LIN {X 0,Y 362.034,Z 645.085,A -85,B 0,C 180,E1 -21360.313,E2 -21360.313} C_VEL
LIN {X 0,Y 359.449,Z 640.545,A -85,B 0,C 180,E1 -21361.106,E2 -21361.106} C_VEL
LIN {X 0,Y 359.251,Z 639.964,A -85,B 0,C 180,E1 -21361.22,E2 -21361.22} C_VEL
LIN {X 0,Y 357.675,Z 633.23,A -85,B 0,C 180,E1 -21364.664,E2 -21364.664} C_VEL
LIN {X 0,Y 356.244,Z 627.609,A -85,B 0,C 180,E1 -21368.142,E2 -21368.142} C_VEL
LIN {X 0,Y 354.982,Z 623.589,A -85,B 0,C 180,E1 -21371.426,E2 -21371.426} C_VEL
LIN {X 0,Y 354.115,Z 620.735,A -85,B 0,C 180,E1 -21374.595,E2 -21374.595} C_VEL
LIN {X 0,Y 353.624,Z 618.917,A -85,B 0,C 180,E1 -21377.665,E2 -21377.665} C_VEL
LIN {X 0,Y 353.31,Z 618.175,A -85,B 0,C 180,E1 -21380.641,E2 -21380.641} C_VEL
LIN {X 0,Y 353.46,Z 618.481,A -85,B 0,C 180,E1 -21384.34,E2 -21384.34} C_VEL
LIN {X 0,Y 353.86,Z 619.974,A -85,B 0,C 180,E1 -21387.693,E2 -21387.693} C_VEL
LIN {X 0,Y 354.531,Z 621.978,A -85,B 0,C 180,E1 -21390.401,E2 -21390.401} C_VEL
LIN {X 0,Y 355.324,Z 624.648,A -85,B 0,C 180,E1 -21393.038,E2 -21393.038} C_VEL
LIN {X 0,Y 356.135,Z 627.934,A -85,B 0,C 180,E1 -21395.605,E2 -21395.605} C_VEL
LIN {X 0,Y 357.351,Z 632.416,A -85,B 0,C 180,E1 -21398.474,E2 -21398.474} C_VEL
LIN {X 0,Y 359.745,Z 636.348,A -85,B 0,C 180,E1 -21399.232,E2 -21399.232} C_VEL
LIN {X 0,Y 361.184,Z 638.274,A -85,B 0,C 180,E1 -21399.647,E2 -21399.647} C_VEL
LIN {X 0,Y 364.586,Z 643.755,A -85,B 0,C 180,E1 -21400.618,E2 -21400.618} C_VEL
LIN {X 0,Y 369.272,Z 651.818,A -85,B 0,C 180,E1 -21401.891,E2 -21401.891} C_VEL
LIN {X 0,Y 374.557,Z 662.104,A -85,B 0,C 180,E1 -21403.232,E2 -21403.232} C_VEL
LIN {X 0,Y 377.698,Z 669.576,A -85,B 0,C 180,E1 -21404.051,E2 -21404.051} C_VEL
LIN {X 0,Y 378.425,Z 674.581,A -85,B 0,C 180,E1 -21404.369,E2 -21404.369} C_VEL
LIN {X 0,Y 373.198,Z 737.25,A -85,B 0,C 180,E1 -21406.258,E2 -21406.258} C_VEL
LIN {X 0,Y 372.142,Z 747.157,A -85,B 0,C 180,E1 -21406.669,E2 -21406.669} C_VEL
LIN {X 0,Y 370.881,Z 756.699,A -85,B 0,C 180,E1 -21407.178,E2 -21407.178} C_VEL
LIN {X 0,Y 369.456,Z 766.257,A -85,B 0,C 180,E1 -21407.824,E2 -21407.824} C_VEL
LIN {X 0,Y 367.532,Z 777.167,A -85,B 0,C 180,E1 -21408.735,E2 -21408.735} C_VEL
LIN {X 0,Y 365.707,Z 786.264,A -85,B 0,C 180,E1 -21409.656,E2 -21409.656} C_VEL
LIN {X 0,Y 364.062,Z 793.981,A -85,B 0,C 180,E1 -21410.587,E2 -21410.587} C_VEL
LIN {X 0,Y 362.212,Z 801.591,A -85,B 0,C 180,E1 -21411.66,E2 -21411.66} C_VEL
LIN {X 0,Y 360.099,Z 809.415,A -85,B 0,C 180,E1 -21412.984,E2 -21412.984} C_VEL
LIN {X 0,Y 358.035,Z 816.293,A -85,B 0,C 180,E1 -21414.386,E2 -21414.386} C_VEL
LIN {X 0,Y 356.572,Z 820.935,A -85,B 0,C 180,E1 -21415.493,E2 -21415.493} C_VEL
LIN {X 0,Y 354.669,Z 826.661,A -85,B 0,C 180,E1 -21417.17,E2 -21417.17} C_VEL
LIN {X 0,Y 353.04,Z 831.154,A -85,B 0,C 180,E1 -21418.863,E2 -21418.863} C_VEL
LIN {X 0,Y 352.202,Z 833.462,A -85,B 0,C 180,E1 -21420,E2 -21420} C_VEL
LIN {X 0,Y 350.875,Z 836.886,A -85,B 0,C 180,E1 -21422.288,E2 -21422.288} C_VEL
LIN {X 0,Y 349.954,Z 838.441,A -85,B 0,C 180,E1 -21424.592,E2 -21424.592} C_VEL
LIN {X 0,Y 349.611,Z 838.707,A -85,B 0,C 180,E1 -21425.749,E2 -21425.749} C_VEL
LIN {X 0,Y 349.177,Z 837.732,A -85,B 0,C 180,E1 -21428.072,E2 -21428.072} C_VEL
LIN {X 0,Y 349.123,Z 836.645,A -85,B 0,C 180,E1 -21429.236,E2 -21429.236} C_VEL
LIN {X 0,Y 349.169,Z 834.725,A -85,B 0,C 180,E1 -21430.592,E2 -21430.592} C_VEL
LIN {X 0,Y 349.117,Z 831.765,A -85,B 0,C 180,E1 -21432.161,E2 -21432.161} C_VEL
LIN {X 0,Y 349.316,Z 827.362,A -85,B 0,C 180,E1 -21433.923,E2 -21433.923} C_VEL
LIN {X 0,Y 349.612,Z 822.276,A -85,B 0,C 180,E1 -21435.516,E2 -21435.516} C_VEL
LIN {X 0,Y 349.838,Z 816.988,A -85,B 0,C 180,E1 -21436.877,E2 -21436.877} C_VEL
LIN {X 0,Y 350.091,Z 811.586,A -85,B 0,C 180,E1 -21438.066,E2 -21438.066} C_VEL
LIN {X 0,Y 350.483,Z 805.301,A -85,B 0,C 180,E1 -21439.253,E2 -21439.253} C_VEL
LIN {X 0,Y 350.964,Z 797.406,A -85,B 0,C 180,E1 -21440.512,E2 -21440.512} C_VEL
LIN {X 0,Y 351.517,Z 787.781,A -85,B 0,C 180,E1 -21441.785,E2 -21441.785} C_VEL
LIN {X 0,Y 352.089,Z 778.326,A -85,B 0,C 180,E1 -21442.825,E2 -21442.825} C_VEL
LIN {X 0,Y 352.732,Z 767.619,A -85,B 0,C 180,E1 -21443.791,E2 -21443.791} C_VEL
LIN {X 0,Y 353.212,Z 757.652,A -85,B 0,C 180,E1 -21444.521,E2 -21444.521} C_VEL
LIN {X 0,Y 353.539,Z 747.147,A -85,B 0,C 180,E1 -21445.133,E2 -21445.133} C_VEL
LIN {X 0,Y 353.943,Z 736.192,A -85,B 0,C 180,E1 -21445.612,E2 -21445.612} C_VEL
LIN {X 0,Y 354.734,Z 713.298,A -85,B 0,C 180,E1 -21446.298,E2 -21446.298} C_VEL
LIN {X 0,Y 356.077,Z 658.366,A -85,B 0,C 180,E1 -21447.873,E2 -21447.873} C_VEL
LIN {X 0,Y 353.084,Z 631.016,A -85,B 0,C 180,E1 -21448.746,E2 -21448.746} C_VEL
LIN {X 0,Y 352.843,Z 627.653,A -85,B 0,C 180,E1 -21448.863,E2 -21448.863} C_VEL
LIN {X 0,Y 353.374,Z 621.195,A -85,B 0,C 180,E1 -21450.69,E2 -21450.69} C_VEL
LIN {X 0,Y 352.052,Z 613.561,A -85,B 0,C 180,E1 -21452.992,E2 -21452.992} C_VEL
LIN {X 0,Y 351.912,Z 613.577,A -85,B 0,C 180,E1 -21457.235,E2 -21457.235} C_VEL
LIN {X 0,Y 351.881,Z 613.582,A -85,B 0,C 180,E1 -21461.062,E2 -21461.062} C_VEL
LIN {X 0,Y 351.929,Z 613.579,A -85,B 0,C 180,E1 -21464.233,E2 -21464.233} C_VEL
LIN {X 0,Y 351.919,Z 613.577,A -85,B 0,C 180,E1 -21467.427,E2 -21467.427} C_VEL
LIN {X 0,Y 351.872,Z 613.583,A -85,B 0,C 180,E1 -21470.926,E2 -21470.926} C_VEL
LIN {X 0,Y 351.907,Z 613.579,A -85,B 0,C 180,E1 -21473.335,E2 -21473.335} C_VEL
LIN {X 0,Y 351.883,Z 613.581,A -85,B 0,C 180,E1 -21476.723,E2 -21476.723} C_VEL
LIN {X 0,Y 351.923,Z 613.582,A -85,B 0,C 180,E1 -21480.159,E2 -21480.159} C_VEL
LIN {X 0,Y 351.926,Z 613.578,A -85,B 0,C 180,E1 -21483.59,E2 -21483.59} C_VEL
LIN {X 0,Y 351.975,Z 613.571,A -85,B 0,C 180,E1 -21486.546,E2 -21486.546} C_VEL
LIN {X 0,Y 351.959,Z 613.576,A -85,B 0,C 180,E1 -21490.225,E2 -21490.225} C_VEL
LIN {X 0,Y 352.021,Z 613.569,A -85,B 0,C 180,E1 -21493.825,E2 -21493.825} C_VEL
LIN {X 0,Y 352.11,Z 613.554,A -85,B 0,C 180,E1 -21497.36,E2 -21497.36} C_VEL
LIN {X 0,Y 352.152,Z 613.549,A -85,B 0,C 180,E1 -21500.844,E2 -21500.844} C_VEL
LIN {X 0,Y 352.258,Z 613.537,A -85,B 0,C 180,E1 -21504.294,E2 -21504.294} C_VEL
LIN {X 0,Y 352.315,Z 613.531,A -85,B 0,C 180,E1 -21507.721,E2 -21507.721} C_VEL
LIN {X 0,Y 352.255,Z 613.536,A -85,B 0,C 180,E1 -21511.139,E2 -21511.139} C_VEL
LIN {X 0,Y 352.328,Z 613.526,A -85,B 0,C 180,E1 -21514.561,E2 -21514.561} C_VEL
LIN {X 0,Y 352.244,Z 613.537,A -85,B 0,C 180,E1 -21516.852,E2 -21516.852} C_VEL
LIN {X 0,Y 352.1,Z 613.558,A -85,B 0,C 180,E1 -21520.314,E2 -21520.314} C_VEL
LIN {X 0,Y 352.044,Z 613.565,A -85,B 0,C 180,E1 -21523.813,E2 -21523.813} C_VEL
LIN {X 0,Y 352.014,Z 613.566,A -85,B 0,C 180,E1 -21527.366,E2 -21527.366} C_VEL
LIN {X 0,Y 351.956,Z 613.573,A -85,B 0,C 180,E1 -21530.991,E2 -21530.991} C_VEL
LIN {X 0,Y 351.941,Z 613.577,A -85,B 0,C 180,E1 -21533.724,E2 -21533.724} C_VEL
LIN {X 0,Y 351.908,Z 613.579,A -85,B 0,C 180,E1 -21537.245,E2 -21537.245} C_VEL
LIN {X 0,Y 351.926,Z 613.581,A -85,B 0,C 180,E1 -21539.84,E2 -21539.84} C_VEL
LIN {X 0,Y 351.92,Z 613.581,A -85,B 0,C 180,E1 -21543.869,E2 -21543.869} C_VEL
LIN {X 0,Y 351.953,Z 613.573,A -85,B 0,C 180,E1 -21547.245,E2 -21547.245} C_VEL
LIN {X 0,Y 351.92,Z 613.577,A -85,B 0,C 180,E1 -21551.057,E2 -21551.057} C_VEL
LIN {X 0,Y 351.927,Z 613.579,A -85,B 0,C 180,E1 -21554.234,E2 -21554.234} C_VEL
LIN {X 0,Y 351.918,Z 613.578,A -85,B 0,C 180,E1 -21557.428,E2 -21557.428} C_VEL
LIN {X 0,Y 351.899,Z 613.58,A -85,B 0,C 180,E1 -21560.921,E2 -21560.921} C_VEL
LIN {X 0,Y 351.933,Z 613.575,A -85,B 0,C 180,E1 -21564.688,E2 -21564.688} C_VEL
LIN {X 0,Y 351.92,Z 613.577,A -85,B 0,C 180,E1 -21568.853,E2 -21568.853} C_VEL
LIN {X 0,Y 351.96,Z 613.573,A -85,B 0,C 180,E1 -21571.47,E2 -21571.47} C_VEL
LIN {X 0,Y 351.9,Z 613.58,A -85,B 0,C 180,E1 -21575.292,E2 -21575.292} C_VEL
LIN {X 0,Y 351.907,Z 613.583,A -85,B 0,C 180,E1 -21577.78,E2 -21577.78} C_VEL
LIN {X 0,Y 351.958,Z 613.576,A -85,B 0,C 180,E1 -21580.226,E2 -21580.226} C_VEL
LIN {X 0,Y 351.98,Z 613.573,A -85,B 0,C 180,E1 -21583.824,E2 -21583.824} C_VEL
LIN {X 0,Y 352.108,Z 613.555,A -85,B 0,C 180,E1 -21587.361,E2 -21587.361} C_VEL
LIN {X 0,Y 352.156,Z 613.547,A -85,B 0,C 180,E1 -21590.845,E2 -21590.845} C_VEL
LIN {X 0,Y 352.3,Z 613.533,A -85,B 0,C 180,E1 -21594.295,E2 -21594.295} C_VEL
LIN {X 0,Y 352.319,Z 613.531,A -85,B 0,C 180,E1 -21597.722,E2 -21597.722} C_VEL
LIN {X 0,Y 352.255,Z 613.535,A -85,B 0,C 180,E1 -21601.14,E2 -21601.14} C_VEL
LIN {X 0,Y 352.327,Z 613.528,A -85,B 0,C 180,E1 -21604.561,E2 -21604.561} C_VEL
LIN {X 0,Y 352.248,Z 613.537,A -85,B 0,C 180,E1 -21606.853,E2 -21606.853} C_VEL
LIN {X 0,Y 352.181,Z 613.551,A -85,B 0,C 180,E1 -21608.003,E2 -21608.003} C_VEL
LIN {X 0,Y 351.48,Z 613.633,A -85,B 0,C 180,E1 -21608.957,E2 -21608.957} C_VEL
LIN {X 0,Y 348.656,Z 613.984,A -85,B 0,C 180,E1 -21610.508,E2 -21610.508} C_VEL
LIN {X 0,Y 346.248,Z 614.287,A -85,B 0,C 180,E1 -21611.763,E2 -21611.763} C_VEL
LIN {X 0,Y 345.156,Z 614.419,A -85,B 0,C 180,E1 -21612.733,E2 -21612.733} C_VEL
LIN {X 0,Y 345.035,Z 614.434,A -85,B 0,C 180,E1 -21613.062,E2 -21613.062} C_VEL
LIN {X 0,Y 344.905,Z 614.452,A -85,B 0,C 180,E1 -21617.352,E2 -21617.352} C_VEL
LIN {X 0,Y 344.874,Z 614.454,A -85,B 0,C 180,E1 -21620.89,E2 -21620.89} C_VEL
LIN {X 0,Y 344.883,Z 614.459,A -85,B 0,C 180,E1 -21623.966,E2 -21623.966} C_VEL
LIN {X 0,Y 344.893,Z 614.457,A -85,B 0,C 180,E1 -21627.847,E2 -21627.847} C_VEL
LIN {X 0,Y 344.816,Z 614.462,A -85,B 0,C 180,E1 -21631.442,E2 -21631.442} C_VEL
LIN {X 0,Y 344.834,Z 614.461,A -85,B 0,C 180,E1 -21634.663,E2 -21634.663} C_VEL
LIN {X 0,Y 344.854,Z 614.46,A -85,B 0,C 180,E1 -21637.614,E2 -21637.614} C_VEL
LIN {X 0,Y 344.822,Z 614.46,A -85,B 0,C 180,E1 -21641.272,E2 -21641.272} C_VEL
LIN {X 0,Y 344.799,Z 614.465,A -85,B 0,C 180,E1 -21644.683,E2 -21644.683} C_VEL
LIN {X 0,Y 344.817,Z 614.467,A -85,B 0,C 180,E1 -21647.907,E2 -21647.907} C_VEL
LIN {X 0,Y 344.81,Z 614.461,A -85,B 0,C 180,E1 -21650.97,E2 -21650.97} C_VEL
LIN {X 0,Y 344.821,Z 614.464,A -85,B 0,C 180,E1 -21654.344,E2 -21654.344} C_VEL
LIN {X 0,Y 344.826,Z 614.461,A -85,B 0,C 180,E1 -21656.739,E2 -21656.739} C_VEL
LIN {X 0,Y 344.833,Z 614.458,A -85,B 0,C 180,E1 -21660.824,E2 -21660.824} C_VEL
LIN {X 0,Y 344.968,Z 614.643,A -85,B 0,C 180,E1 -21663.175,E2 -21663.175} C_VEL
LIN {X 0,Y 347.071,Z 626.547,A -85,B 0,C 180,E1 -21666.51,E2 -21666.51} C_VEL
LIN {X 0,Y 347.053,Z 630.044,A -85,B 0,C 180,E1 -21667.451,E2 -21667.451} C_VEL
LIN {X 0,Y 345.418,Z 643.632,A -85,B 0,C 180,E1 -21670.991,E2 -21670.991} C_VEL
LIN {X 0,Y 347.217,Z 668.999,A -85,B 0,C 180,E1 -21671.803,E2 -21671.803} C_VEL
LIN {X 0,Y 348.767,Z 684.999,A -85,B 0,C 180,E1 -21672.312,E2 -21672.312} C_VEL
LIN {X 0,Y 347.023,Z 749.499,A -85,B 0,C 180,E1 -21674.225,E2 -21674.225} C_VEL
LIN {X 0,Y 346.578,Z 759.945,A -85,B 0,C 180,E1 -21674.655,E2 -21674.655} C_VEL
LIN {X 0,Y 346.235,Z 769.907,A -85,B 0,C 180,E1 -21675.202,E2 -21675.202} C_VEL
LIN {X 0,Y 345.748,Z 780.31,A -85,B 0,C 180,E1 -21675.93,E2 -21675.93} C_VEL
LIN {X 0,Y 345.259,Z 789.479,A -85,B 0,C 180,E1 -21676.716,E2 -21676.716} C_VEL
LIN {X 0,Y 344.524,Z 799.727,A -85,B 0,C 180,E1 -21677.789,E2 -21677.789} C_VEL
LIN {X 0,Y 344.029,Z 808.158,A -85,B 0,C 180,E1 -21678.848,E2 -21678.848} C_VEL
LIN {X 0,Y 343.55,Z 816.054,A -85,B 0,C 180,E1 -21680.02,E2 -21680.02} C_VEL
LIN {X 0,Y 343.024,Z 824.278,A -85,B 0,C 180,E1 -21681.487,E2 -21681.487} C_VEL
LIN {X 0,Y 342.777,Z 831.149,A -85,B 0,C 180,E1 -21682.958,E2 -21682.958} C_VEL
LIN {X 0,Y 342.591,Z 835.863,A -85,B 0,C 180,E1 -21684.133,E2 -21684.133} C_VEL
LIN {X 0,Y 342.46,Z 841.572,A -85,B 0,C 180,E1 -21685.895,E2 -21685.895} C_VEL
LIN {X 0,Y 342.421,Z 846.02,A -85,B 0,C 180,E1 -21687.656,E2 -21687.656} C_VEL
LIN {X 0,Y 342.371,Z 848.381,A -85,B 0,C 180,E1 -21688.828,E2 -21688.828} C_VEL
LIN {X 0,Y 342.277,Z 851.57,A -85,B 0,C 180,E1 -21691.173,E2 -21691.173} C_VEL
LIN {X 0,Y 342.251,Z 852.514,A -85,B 0,C 180,E1 -21692.346,E2 -21692.346} C_VEL
LIN {X 0,Y 342.314,Z 853.154,A -85,B 0,C 180,E1 -21694.695,E2 -21694.695} C_VEL
LIN {X 0,Y 342.824,Z 852.017,A -85,B 0,C 180,E1 -21697.042,E2 -21697.042} C_VEL
LIN {X 0,Y 343.184,Z 850.939,A -85,B 0,C 180,E1 -21698.214,E2 -21698.214} C_VEL
LIN {X 0,Y 344.459,Z 847.292,A -85,B 0,C 180,E1 -21700.545,E2 -21700.545} C_VEL
LIN {X 0,Y 345.803,Z 843.392,A -85,B 0,C 180,E1 -21702.28,E2 -21702.28} C_VEL
LIN {X 0,Y 347.54,Z 838.373,A -85,B 0,C 180,E1 -21703.996,E2 -21703.996} C_VEL
LIN {X 0,Y 349.51,Z 832.307,A -85,B 0,C 180,E1 -21705.651,E2 -21705.651} C_VEL
LIN {X 0,Y 351.436,Z 825.979,A -85,B 0,C 180,E1 -21707.067,E2 -21707.067} C_VEL
LIN {X 0,Y 353.704,Z 818.316,A -85,B 0,C 180,E1 -21708.473,E2 -21708.473} C_VEL
LIN {X 0,Y 356.07,Z 809.306,A -85,B 0,C 180,E1 -21709.837,E2 -21709.837} C_VEL
LIN {X 0,Y 358.245,Z 800.757,A -85,B 0,C 180,E1 -21710.906,E2 -21710.906} C_VEL
LIN {X 0,Y 360.206,Z 792.083,A -85,B 0,C 180,E1 -21711.833,E2 -21711.833} C_VEL
LIN {X 0,Y 362.445,Z 781.582,A -85,B 0,C 180,E1 -21712.738,E2 -21712.738} C_VEL
LIN {X 0,Y 364.311,Z 771.526,A -85,B 0,C 180,E1 -21713.438,E2 -21713.438} C_VEL
LIN {X 0,Y 365.885,Z 761.383,A -85,B 0,C 180,E1 -21714.005,E2 -21714.005} C_VEL
LIN {X 0,Y 367.204,Z 750.541,A -85,B 0,C 180,E1 -21714.475,E2 -21714.475} C_VEL
LIN {X 0,Y 369.726,Z 721.521,A -85,B 0,C 180,E1 -21715.381,E2 -21715.381} C_VEL
LIN {X 0,Y 371.831,Z 694.493,A -85,B 0,C 180,E1 -21716.242,E2 -21716.242} C_VEL
LIN {X 0,Y 369.906,Z 680.185,A -85,B 0,C 180,E1 -21717.182,E2 -21717.182} C_VEL
LIN {X 0,Y 367.596,Z 668.954,A -85,B 0,C 180,E1 -21718.08,E2 -21718.08} C_VEL
LIN {X 0,Y 363.48,Z 660.04,A -85,B 0,C 180,E1 -21719.265,E2 -21719.265} C_VEL
LIN {X 0,Y 360.148,Z 653.811,A -85,B 0,C 180,E1 -21720.22,E2 -21720.22} C_VEL
LIN {X 0,Y 358.168,Z 650.178,A -85,B 0,C 180,E1 -21720.835,E2 -21720.835} C_VEL
LIN {X 0,Y 355.269,Z 645.127,A -85,B 0,C 180,E1 -21721.761,E2 -21721.761} C_VEL
LIN {X 0,Y 352.46,Z 640.727,A -85,B 0,C 180,E1 -21722.694,E2 -21722.694} C_VEL
LIN {X 0,Y 352.039,Z 639.672,A -85,B 0,C 180,E1 -21722.876,E2 -21722.876} C_VEL
LIN {X 0,Y 351.049,Z 635.18,A -85,B 0,C 180,E1 -21725.355,E2 -21725.355} C_VEL
LIN {X 0,Y 349.749,Z 630.253,A -85,B 0,C 180,E1 -21728.643,E2 -21728.643} C_VEL
LIN {X 0,Y 348.608,Z 626.433,A -85,B 0,C 180,E1 -21731.976,E2 -21731.976} C_VEL
LIN {X 0,Y 347.789,Z 623.782,A -85,B 0,C 180,E1 -21735.179,E2 -21735.179} C_VEL
LIN {X 0,Y 347.365,Z 622.183,A -85,B 0,C 180,E1 -21738.285,E2 -21738.285} C_VEL
LIN {X 0,Y 347.118,Z 621.655,A -85,B 0,C 180,E1 -21741.904,E2 -21741.904} C_VEL
LIN {X 0,Y 347.254,Z 621.942,A -85,B 0,C 180,E1 -21744.2,E2 -21744.2} C_VEL
LIN {X 0,Y 347.55,Z 623.069,A -85,B 0,C 180,E1 -21747.033,E2 -21747.033} C_VEL
LIN {X 0,Y 348.152,Z 624.946,A -85,B 0,C 180,E1 -21749.896,E2 -21749.896} C_VEL
LIN {X 0,Y 348.868,Z 627.364,A -85,B 0,C 180,E1 -21752.497,E2 -21752.497} C_VEL
LIN {X 0,Y 349.627,Z 630.504,A -85,B 0,C 180,E1 -21755.12,E2 -21755.12} C_VEL
LIN {X 0,Y 350.23,Z 632.802,A -85,B 0,C 180,E1 -21756.734,E2 -21756.734} C_VEL
LIN {X 0,Y 352.999,Z 637.077,A -85,B 0,C 180,E1 -21757.724,E2 -21757.724} C_VEL
LIN {X 0,Y 354.289,Z 638.717,A -85,B 0,C 180,E1 -21758.14,E2 -21758.14} C_VEL
LIN {X 0,Y 357.077,Z 642.881,A -85,B 0,C 180,E1 -21759.021,E2 -21759.021} C_VEL
LIN {X 0,Y 361.209,Z 649.783,A -85,B 0,C 180,E1 -21760.281,E2 -21760.281} C_VEL
LIN {X 0,Y 365.313,Z 656.876,A -85,B 0,C 180,E1 -21761.422,E2 -21761.422} C_VEL
LIN {X 0,Y 370.195,Z 666.732,A -85,B 0,C 180,E1 -21762.745,E2 -21762.745} C_VEL
LIN {X 0,Y 372.868,Z 673.14,A -85,B 0,C 180,E1 -21763.464,E2 -21763.464} C_VEL
LIN {X 0,Y 373.23,Z 676.01,A -85,B 0,C 180,E1 -21763.65,E2 -21763.65} C_VEL
LIN {X 0,Y 367.703,Z 738.471,A -85,B 0,C 180,E1 -21765.591,E2 -21765.591} C_VEL
LIN {X 0,Y 366.47,Z 748.855,A -85,B 0,C 180,E1 -21766.036,E2 -21766.036} C_VEL
LIN {X 0,Y 365.207,Z 758.036,A -85,B 0,C 180,E1 -21766.552,E2 -21766.552} C_VEL
LIN {X 0,Y 363.706,Z 767.404,A -85,B 0,C 180,E1 -21767.204,E2 -21767.204} C_VEL
LIN {X 0,Y 361.955,Z 776.745,A -85,B 0,C 180,E1 -21767.993,E2 -21767.993} C_VEL
LIN {X 0,Y 360.051,Z 785.832,A -85,B 0,C 180,E1 -21768.924,E2 -21768.924} C_VEL
LIN {X 0,Y 358.264,Z 793.592,A -85,B 0,C 180,E1 -21769.865,E2 -21769.865} C_VEL
LIN {X 0,Y 355.804,Z 802.97,A -85,B 0,C 180,E1 -21771.224,E2 -21771.224} C_VEL
LIN {X 0,Y 353.662,Z 810.45,A -85,B 0,C 180,E1 -21772.535,E2 -21772.535} C_VEL
LIN {X 0,Y 351.865,Z 816.176,A -85,B 0,C 180,E1 -21773.714,E2 -21773.714} C_VEL
LIN {X 0,Y 350.324,Z 820.846,A -85,B 0,C 180,E1 -21774.838,E2 -21774.838} C_VEL
LIN {X 0,Y 348.231,Z 826.61,A -85,B 0,C 180,E1 -21776.54,E2 -21776.54} C_VEL
LIN {X 0,Y 346.498,Z 831.131,A -85,B 0,C 180,E1 -21778.262,E2 -21778.262} C_VEL
LIN {X 0,Y 345.127,Z 834.576,A -85,B 0,C 180,E1 -21780,E2 -21780} C_VEL
LIN {X 0,Y 343.773,Z 837.485,A -85,B 0,C 180,E1 -21782.335,E2 -21782.335} C_VEL
LIN {X 0,Y 343.284,Z 838.411,A -85,B 0,C 180,E1 -21783.509,E2 -21783.509} C_VEL
LIN {X 0,Y 342.468,Z 838.801,A -85,B 0,C 180,E1 -21785.869,E2 -21785.869} C_VEL
LIN {X 0,Y 342.193,Z 838.395,A -85,B 0,C 180,E1 -21787.054,E2 -21787.054} C_VEL
LIN {X 0,Y 342.038,Z 836.267,A -85,B 0,C 180,E1 -21789.429,E2 -21789.429} C_VEL
LIN {X 0,Y 342.024,Z 833.458,A -85,B 0,C 180,E1 -21791.218,E2 -21791.218} C_VEL
LIN {X 0,Y 342.117,Z 829.515,A -85,B 0,C 180,E1 -21793.015,E2 -21793.015} C_VEL
LIN {X 0,Y 342.393,Z 824.32,A -85,B 0,C 180,E1 -21794.816,E2 -21794.816} C_VEL
LIN {X 0,Y 342.642,Z 819.201,A -85,B 0,C 180,E1 -21796.26,E2 -21796.26} C_VEL
LIN {X 0,Y 342.956,Z 812.368,A -85,B 0,C 180,E1 -21797.839,E2 -21797.839} C_VEL
LIN {X 0,Y 343.433,Z 804.407,A -85,B 0,C 180,E1 -21799.355,E2 -21799.355} C_VEL
LIN {X 0,Y 343.932,Z 796.211,A -85,B 0,C 180,E1 -21800.659,E2 -21800.659} C_VEL
LIN {X 0,Y 344.418,Z 787.823,A -85,B 0,C 180,E1 -21801.786,E2 -21801.786} C_VEL
LIN {X 0,Y 345.005,Z 778.404,A -85,B 0,C 180,E1 -21802.847,E2 -21802.847} C_VEL
LIN {X 0,Y 345.585,Z 768.709,A -85,B 0,C 180,E1 -21803.755,E2 -21803.755} C_VEL
LIN {X 0,Y 346.092,Z 758.397,A -85,B 0,C 180,E1 -21804.539,E2 -21804.539} C_VEL
LIN {X 0,Y 346.445,Z 748.079,A -85,B 0,C 180,E1 -21805.163,E2 -21805.163} C_VEL
LIN {X 0,Y 346.876,Z 736.395,A -85,B 0,C 180,E1 -21805.69,E2 -21805.69} C_VEL
LIN {X 0,Y 347.743,Z 709.759,A -85,B 0,C 180,E1 -21806.505,E2 -21806.505} C_VEL
LIN {X 0,Y 349.04,Z 658.977,A -85,B 0,C 180,E1 -21807.996,E2 -21807.996} C_VEL
LIN {X 0,Y 346.07,Z 631.768,A -85,B 0,C 180,E1 -21808.884,E2 -21808.884} C_VEL
LIN {X 0,Y 345.801,Z 627.845,A -85,B 0,C 180,E1 -21809.022,E2 -21809.022} C_VEL
LIN {X 0,Y 346.311,Z 622.063,A -85,B 0,C 180,E1 -21810.689,E2 -21810.689} C_VEL
LIN {X 0,Y 345.021,Z 614.437,A -85,B 0,C 180,E1 -21812.978,E2 -21812.978} C_VEL
LIN {X 0,Y 344.859,Z 614.461,A -85,B 0,C 180,E1 -21816.087,E2 -21816.087} C_VEL
LIN {X 0,Y 344.818,Z 614.463,A -85,B 0,C 180,E1 -21819.474,E2 -21819.474} C_VEL
LIN {X 0,Y 344.854,Z 614.457,A -85,B 0,C 180,E1 -21823.012,E2 -21823.012} C_VEL
LIN {X 0,Y 344.861,Z 614.458,A -85,B 0,C 180,E1 -21826.324,E2 -21826.324} C_VEL
LIN {X 0,Y 344.813,Z 614.464,A -85,B 0,C 180,E1 -21829.455,E2 -21829.455} C_VEL
LIN {X 0,Y 344.849,Z 614.46,A -85,B 0,C 180,E1 -21832.457,E2 -21832.457} C_VEL
LIN {X 0,Y 344.839,Z 614.459,A -85,B 0,C 180,E1 -21835.337,E2 -21835.337} C_VEL
LIN {X 0,Y 344.866,Z 614.457,A -85,B 0,C 180,E1 -21838.543,E2 -21838.543} C_VEL
LIN {X 0,Y 344.892,Z 614.457,A -85,B 0,C 180,E1 -21842.153,E2 -21842.153} C_VEL
LIN {X 0,Y 344.89,Z 614.458,A -85,B 0,C 180,E1 -21846.05,E2 -21846.05} C_VEL
LIN {X 0,Y 344.929,Z 614.452,A -85,B 0,C 180,E1 -21849.805,E2 -21849.805} C_VEL
LIN {X 0,Y 344.975,Z 614.443,A -85,B 0,C 180,E1 -21853.485,E2 -21853.485} C_VEL
LIN {X 0,Y 345.097,Z 614.426,A -85,B 0,C 180,E1 -21857.099,E2 -21857.099} C_VEL
LIN {X 0,Y 345.092,Z 614.429,A -85,B 0,C 180,E1 -21860.655,E2 -21860.655} C_VEL
LIN {X 0,Y 345.23,Z 614.413,A -85,B 0,C 180,E1 -21864.177,E2 -21864.177} C_VEL
LIN {X 0,Y 345.275,Z 614.407,A -85,B 0,C 180,E1 -21867.674,E2 -21867.674} C_VEL
LIN {X 0,Y 345.23,Z 614.411,A -85,B 0,C 180,E1 -21871.162,E2 -21871.162} C_VEL
LIN {X 0,Y 345.284,Z 614.403,A -85,B 0,C 180,E1 -21874.654,E2 -21874.654} C_VEL
LIN {X 0,Y 345.205,Z 614.413,A -85,B 0,C 180,E1 -21876.993,E2 -21876.993} C_VEL
LIN {X 0,Y 345.042,Z 614.435,A -85,B 0,C 180,E1 -21880.527,E2 -21880.527} C_VEL
LIN {X 0,Y 345.083,Z 614.428,A -85,B 0,C 180,E1 -21883.022,E2 -21883.022} C_VEL
LIN {X 0,Y 344.978,Z 614.443,A -85,B 0,C 180,E1 -21887.393,E2 -21887.393} C_VEL
LIN {X 0,Y 344.901,Z 614.453,A -85,B 0,C 180,E1 -21891.441,E2 -21891.441} C_VEL
LIN {X 0,Y 344.865,Z 614.455,A -85,B 0,C 180,E1 -21895.247,E2 -21895.247} C_VEL
LIN {X 0,Y 344.879,Z 614.455,A -85,B 0,C 180,E1 -21899.172,E2 -21899.172} C_VEL
LIN {X 0,Y 344.864,Z 614.461,A -85,B 0,C 180,E1 -21901.876,E2 -21901.876} C_VEL
LIN {X 0,Y 344.93,Z 614.45,A -85,B 0,C 180,E1 -21905.682,E2 -21905.682} C_VEL
LIN {X 0,Y 344.872,Z 614.455,A -85,B 0,C 180,E1 -21909.022,E2 -21909.022} C_VEL
LIN {X 0,Y 344.862,Z 614.461,A -85,B 0,C 180,E1 -21912.087,E2 -21912.087} C_VEL
LIN {X 0,Y 344.855,Z 614.457,A -85,B 0,C 180,E1 -21915.307,E2 -21915.307} C_VEL
LIN {X 0,Y 344.874,Z 614.456,A -85,B 0,C 180,E1 -21918.718,E2 -21918.718} C_VEL
LIN {X 0,Y 344.883,Z 614.454,A -85,B 0,C 180,E1 -21922.463,E2 -21922.463} C_VEL
LIN {X 0,Y 344.844,Z 614.459,A -85,B 0,C 180,E1 -21925.339,E2 -21925.339} C_VEL
LIN {X 0,Y 344.868,Z 614.457,A -85,B 0,C 180,E1 -21928.544,E2 -21928.544} C_VEL
LIN {X 0,Y 344.893,Z 614.456,A -85,B 0,C 180,E1 -21932.154,E2 -21932.154} C_VEL
LIN {X 0,Y 344.891,Z 614.459,A -85,B 0,C 180,E1 -21936.051,E2 -21936.051} C_VEL
LIN {X 0,Y 344.93,Z 614.452,A -85,B 0,C 180,E1 -21939.805,E2 -21939.805} C_VEL
LIN {X 0,Y 344.944,Z 614.446,A -85,B 0,C 180,E1 -21943.484,E2 -21943.484} C_VEL
LIN {X 0,Y 345.1,Z 614.427,A -85,B 0,C 180,E1 -21947.1,E2 -21947.1} C_VEL
LIN {X 0,Y 345.096,Z 614.427,A -85,B 0,C 180,E1 -21950.656,E2 -21950.656} C_VEL
LIN {X 0,Y 345.282,Z 614.408,A -85,B 0,C 180,E1 -21954.179,E2 -21954.179} C_VEL
LIN {X 0,Y 345.279,Z 614.408,A -85,B 0,C 180,E1 -21957.675,E2 -21957.675} C_VEL
LIN {X 0,Y 345.231,Z 614.41,A -85,B 0,C 180,E1 -21961.163,E2 -21961.163} C_VEL
LIN {X 0,Y 345.283,Z 614.404,A -85,B 0,C 180,E1 -21964.655,E2 -21964.655} C_VEL
LIN {X 0,Y 345.209,Z 614.413,A -85,B 0,C 180,E1 -21966.993,E2 -21966.993} C_VEL
LIN {X 0,Y 345.046,Z 614.434,A -85,B 0,C 180,E1 -21970.527,E2 -21970.527} C_VEL
LIN {X 0,Y 345.035,Z 614.434,A -85,B 0,C 180,E1 -21973.062,E2 -21973.062} C_VEL
LIN {X 0,Y 344.28,Z 614.535,A -85,B 0,C 180,E1 -21974.034,E2 -21974.034} C_VEL
LIN {X 0,Y 341.398,Z 614.896,A -85,B 0,C 180,E1 -21975.616,E2 -21975.616} C_VEL
LIN {X 0,Y 338.992,Z 615.198,A -85,B 0,C 180,E1 -21976.897,E2 -21976.897} C_VEL
LIN {X 0,Y 337.941,Z 615.325,A -85,B 0,C 180,E1 -21977.887,E2 -21977.887} C_VEL
LIN {X 0,Y 337.841,Z 615.335,A -85,B 0,C 180,E1 -21978.223,E2 -21978.223} C_VEL
LIN {X 0,Y 337.819,Z 615.338,A -85,B 0,C 180,E1 -21981.914,E2 -21981.914} C_VEL
LIN {X 0,Y 337.839,Z 615.333,A -85,B 0,C 180,E1 -21984.498,E2 -21984.498} C_VEL
LIN {X 0,Y 337.841,Z 615.332,A -85,B 0,C 180,E1 -21988.481,E2 -21988.481} C_VEL
LIN {X 0,Y 337.754,Z 615.342,A -85,B 0,C 180,E1 -21992.629,E2 -21992.629} C_VEL
LIN {X 0,Y 337.807,Z 615.341,A -85,B 0,C 180,E1 -21996.034,E2 -21996.034} C_VEL
LIN {X 0,Y 337.773,Z 615.341,A -85,B 0,C 180,E1 -21998.471,E2 -21998.471} C_VEL
LIN {X 0,Y 337.766,Z 615.342,A -85,B 0,C 180,E1 -22001.708,E2 -22001.708} C_VEL
LIN {X 0,Y 337.751,Z 615.342,A -85,B 0,C 180,E1 -22005.162,E2 -22005.162} C_VEL
LIN {X 0,Y 337.774,Z 615.341,A -85,B 0,C 180,E1 -22008.426,E2 -22008.426} C_VEL
LIN {X 0,Y 337.776,Z 615.343,A -85,B 0,C 180,E1 -22012,E2 -22012} C_VEL
LIN {X 0,Y 337.767,Z 615.342,A -85,B 0,C 180,E1 -22014.504,E2 -22014.504} C_VEL
LIN {X 0,Y 337.741,Z 615.344,A -85,B 0,C 180,E1 -22017.37,E2 -22017.37} C_VEL
LIN {X 0,Y 337.817,Z 615.334,A -85,B 0,C 180,E1 -22021.518,E2 -22021.518} C_VEL
LIN {X 0,Y 337.922,Z 615.4,A -85,B 0,C 180,E1 -22023.091,E2 -22023.091} C_VEL
LIN {X 0,Y 340.087,Z 627.851,A -85,B 0,C 180,E1 -22026.642,E2 -22026.642} C_VEL
LIN {X 0,Y 339.689,Z 632.558,A -85,B 0,C 180,E1 -22027.927,E2 -22027.927} C_VEL
LIN {X 0,Y 338.38,Z 643.202,A -85,B 0,C 180,E1 -22030.809,E2 -22030.809} C_VEL
LIN {X 0,Y 339.978,Z 667.25,A -85,B 0,C 180,E1 -22031.598,E2 -22031.598} C_VEL
LIN {X 0,Y 341.687,Z 685.839,A -85,B 0,C 180,E1 -22032.208,E2 -22032.208} C_VEL
LIN {X 0,Y 339.945,Z 749.512,A -85,B 0,C 180,E1 -22034.157,E2 -22034.157} C_VEL
LIN {X 0,Y 339.49,Z 759.803,A -85,B 0,C 180,E1 -22034.595,E2 -22034.595} C_VEL
LIN {X 0,Y 339.12,Z 770.254,A -85,B 0,C 180,E1 -22035.191,E2 -22035.191} C_VEL
LIN {X 0,Y 338.638,Z 780.501,A -85,B 0,C 180,E1 -22035.934,E2 -22035.934} C_VEL
LIN {X 0,Y 338.105,Z 790.463,A -85,B 0,C 180,E1 -22036.828,E2 -22036.828} C_VEL
LIN {X 0,Y 337.425,Z 799.57,A -85,B 0,C 180,E1 -22037.814,E2 -22037.814} C_VEL
LIN {X 0,Y 336.912,Z 808.109,A -85,B 0,C 180,E1 -22038.913,E2 -22038.913} C_VEL
LIN {X 0,Y 336.453,Z 815.994,A -85,B 0,C 180,E1 -22040.11,E2 -22040.11} C_VEL
LIN {X 0,Y 336.013,Z 822.747,A -85,B 0,C 180,E1 -22041.308,E2 -22041.308} C_VEL
LIN {X 0,Y 335.739,Z 829.851,A -85,B 0,C 180,E1 -22042.809,E2 -22042.809} C_VEL
LIN {X 0,Y 335.505,Z 836.754,A -85,B 0,C 180,E1 -22044.609,E2 -22044.609} C_VEL
LIN {X 0,Y 335.411,Z 840.66,A -85,B 0,C 180,E1 -22045.809,E2 -22045.809} C_VEL
LIN {X 0,Y 335.352,Z 845.295,A -85,B 0,C 180,E1 -22047.606,E2 -22047.606} C_VEL
LIN {X 0,Y 335.321,Z 847.664,A -85,B 0,C 180,E1 -22048.803,E2 -22048.803} C_VEL
LIN {X 0,Y 335.191,Z 851.152,A -85,B 0,C 180,E1 -22051.198,E2 -22051.198} C_VEL
LIN {X 0,Y 335.13,Z 852.712,A -85,B 0,C 180,E1 -22053.595,E2 -22053.595} C_VEL
LIN {X 0,Y 335.227,Z 852.97,A -85,B 0,C 180,E1 -22054.795,E2 -22054.795} C_VEL
LIN {X 0,Y 335.757,Z 852.089,A -85,B 0,C 180,E1 -22057.191,E2 -22057.191} C_VEL
LIN {X 0,Y 336.141,Z 851.015,A -85,B 0,C 180,E1 -22058.388,E2 -22058.388} C_VEL
LIN {X 0,Y 337.512,Z 847.69,A -85,B 0,C 180,E1 -22060.765,E2 -22060.765} C_VEL
LIN {X 0,Y 338.905,Z 844.009,A -85,B 0,C 180,E1 -22062.534,E2 -22062.534} C_VEL
LIN {X 0,Y 340.731,Z 839.218,A -85,B 0,C 180,E1 -22064.282,E2 -22064.282} C_VEL
LIN {X 0,Y 343.229,Z 831.868,A -85,B 0,C 180,E1 -22066.329,E2 -22066.329} C_VEL
LIN {X 0,Y 345.256,Z 825.7,A -85,B 0,C 180,E1 -22067.717,E2 -22067.717} C_VEL
LIN {X 0,Y 347.592,Z 818.216,A -85,B 0,C 180,E1 -22069.115,E2 -22069.115} C_VEL
LIN {X 0,Y 350.098,Z 809.343,A -85,B 0,C 180,E1 -22070.495,E2 -22070.495} C_VEL
LIN {X 0,Y 352.373,Z 800.908,A -85,B 0,C 180,E1 -22071.577,E2 -22071.577} C_VEL
LIN {X 0,Y 354.79,Z 790.849,A -85,B 0,C 180,E1 -22072.643,E2 -22072.643} C_VEL
LIN {X 0,Y 356.786,Z 781.826,A -85,B 0,C 180,E1 -22073.425,E2 -22073.425} C_VEL
LIN {X 0,Y 358.909,Z 770.813,A -85,B 0,C 180,E1 -22074.195,E2 -22074.195} C_VEL
LIN {X 0,Y 360.554,Z 760.537,A -85,B 0,C 180,E1 -22074.765,E2 -22074.765} C_VEL
LIN {X 0,Y 361.961,Z 749.684,A -85,B 0,C 180,E1 -22075.236,E2 -22075.236} C_VEL
LIN {X 0,Y 366.714,Z 696.38,A -85,B 0,C 180,E1 -22076.946,E2 -22076.946} C_VEL
LIN {X 0,Y 365.002,Z 683.091,A -85,B 0,C 180,E1 -22077.84,E2 -22077.84} C_VEL
LIN {X 0,Y 363.094,Z 672.965,A -85,B 0,C 180,E1 -22078.678,E2 -22078.678} C_VEL
LIN {X 0,Y 359.032,Z 664.133,A -85,B 0,C 180,E1 -22079.898,E2 -22079.898} C_VEL
LIN {X 0,Y 354.919,Z 656.045,A -85,B 0,C 180,E1 -22081.207,E2 -22081.207} C_VEL
LIN {X 0,Y 351.514,Z 650.252,A -85,B 0,C 180,E1 -22082.324,E2 -22082.324} C_VEL
LIN {X 0,Y 348.845,Z 645.643,A -85,B 0,C 180,E1 -22083.29,E2 -22083.29} C_VEL
LIN {X 0,Y 345.378,Z 640.389,A -85,B 0,C 180,E1 -22084.601,E2 -22084.601} C_VEL
LIN {X 0,Y 344.861,Z 639.187,A -85,B 0,C 180,E1 -22084.882,E2 -22084.882} C_VEL
LIN {X 0,Y 343.836,Z 634.883,A -85,B 0,C 180,E1 -22087.673,E2 -22087.673} C_VEL
LIN {X 0,Y 342.673,Z 630.988,A -85,B 0,C 180,E1 -22090.861,E2 -22090.861} C_VEL
LIN {X 0,Y 341.815,Z 627.967,A -85,B 0,C 180,E1 -22094.175,E2 -22094.175} C_VEL
LIN {X 0,Y 341.227,Z 625.951,A -85,B 0,C 180,E1 -22097.645,E2 -22097.645} C_VEL
LIN {X 0,Y 340.941,Z 625.232,A -85,B 0,C 180,E1 -22100.44,E2 -22100.44} C_VEL
LIN {X 0,Y 340.981,Z 625.284,A -85,B 0,C 180,E1 -22103.436,E2 -22103.436} C_VEL
LIN {X 0,Y 341.254,Z 626.189,A -85,B 0,C 180,E1 -22106.345,E2 -22106.345} C_VEL
LIN {X 0,Y 341.8,Z 627.97,A -85,B 0,C 180,E1 -22109.396,E2 -22109.396} C_VEL
LIN {X 0,Y 342.414,Z 630.133,A -85,B 0,C 180,E1 -22111.934,E2 -22111.934} C_VEL
LIN {X 0,Y 343.235,Z 633.335,A -85,B 0,C 180,E1 -22114.725,E2 -22114.725} C_VEL
LIN {X 0,Y 345.737,Z 637.334,A -85,B 0,C 180,E1 -22115.801,E2 -22115.801} C_VEL
LIN {X 0,Y 347.518,Z 639.403,A -85,B 0,C 180,E1 -22116.45,E2 -22116.45} C_VEL
LIN {X 0,Y 350.604,Z 643.785,A -85,B 0,C 180,E1 -22117.561,E2 -22117.561} C_VEL
LIN {X 0,Y 354.797,Z 650.479,A -85,B 0,C 180,E1 -22118.953,E2 -22118.953} C_VEL
LIN {X 0,Y 359.125,Z 657.818,A -85,B 0,C 180,E1 -22120.295,E2 -22120.295} C_VEL
LIN {X 0,Y 364.473,Z 668.206,A -85,B 0,C 180,E1 -22121.842,E2 -22121.842} C_VEL
LIN {X 0,Y 368.036,Z 676.65,A -85,B 0,C 180,E1 -22122.858,E2 -22122.858} C_VEL
LIN {X 0,Y 366.702,Z 692.894,A -85,B 0,C 180,E1 -22123.398,E2 -22123.398} C_VEL
LIN {X 0,Y 362.394,Z 738.491,A -85,B 0,C 180,E1 -22124.838,E2 -22124.838} C_VEL
LIN {X 0,Y 361.049,Z 749.356,A -85,B 0,C 180,E1 -22125.32,E2 -22125.32} C_VEL
LIN {X 0,Y 359.566,Z 759.374,A -85,B 0,C 180,E1 -22125.906,E2 -22125.906} C_VEL
LIN {X 0,Y 357.976,Z 768.574,A -85,B 0,C 180,E1 -22126.564,E2 -22126.564} C_VEL
LIN {X 0,Y 356.151,Z 777.765,A -85,B 0,C 180,E1 -22127.361,E2 -22127.361} C_VEL
LIN {X 0,Y 354.157,Z 786.743,A -85,B 0,C 180,E1 -22128.304,E2 -22128.304} C_VEL
LIN {X 0,Y 352.011,Z 795.396,A -85,B 0,C 180,E1 -22129.393,E2 -22129.393} C_VEL
LIN {X 0,Y 349.974,Z 802.793,A -85,B 0,C 180,E1 -22130.496,E2 -22130.496} C_VEL
LIN {X 0,Y 347.574,Z 810.606,A -85,B 0,C 180,E1 -22131.89,E2 -22131.89} C_VEL
LIN {X 0,Y 345.378,Z 817.108,A -85,B 0,C 180,E1 -22133.273,E2 -22133.273} C_VEL
LIN {X 0,Y 343.308,Z 822.785,A -85,B 0,C 180,E1 -22134.732,E2 -22134.732} C_VEL
LIN {X 0,Y 341.879,Z 826.599,A -85,B 0,C 180,E1 -22135.888,E2 -22135.888} C_VEL
LIN {X 0,Y 339.965,Z 831.184,A -85,B 0,C 180,E1 -22137.638,E2 -22137.638} C_VEL
LIN {X 0,Y 338.017,Z 835.478,A -85,B 0,C 180,E1 -22140,E2 -22140} C_VEL
LIN {X 0,Y 337.219,Z 837.078,A -85,B 0,C 180,E1 -22141.19,E2 -22141.19} C_VEL
LIN {X 0,Y 336.146,Z 838.79,A -85,B 0,C 180,E1 -22143.584,E2 -22143.584} C_VEL
LIN {X 0,Y 335.667,Z 839.042,A -85,B 0,C 180,E1 -22144.858,E2 -22144.858} C_VEL
LIN {X 0,Y 335.069,Z 838.299,A -85,B 0,C 180,E1 -22147.205,E2 -22147.205} C_VEL
LIN {X 0,Y 334.986,Z 837.219,A -85,B 0,C 180,E1 -22148.416,E2 -22148.416} C_VEL
LIN {X 0,Y 334.957,Z 833.881,A -85,B 0,C 180,E1 -22150.847,E2 -22150.847} C_VEL
LIN {X 0,Y 334.983,Z 830.021,A -85,B 0,C 180,E1 -22152.682,E2 -22152.682} C_VEL
LIN {X 0,Y 335.315,Z 823.881,A -85,B 0,C 180,E1 -22154.826,E2 -22154.826} C_VEL
LIN {X 0,Y 335.556,Z 818.969,A -85,B 0,C 180,E1 -22156.216,E2 -22156.216} C_VEL
LIN {X 0,Y 335.892,Z 811.626,A -85,B 0,C 180,E1 -22157.913,E2 -22157.913} C_VEL
LIN {X 0,Y 336.27,Z 805.293,A -85,B 0,C 180,E1 -22159.151,E2 -22159.151} C_VEL
LIN {X 0,Y 336.832,Z 796.095,A -85,B 0,C 180,E1 -22160.645,E2 -22160.645} C_VEL
LIN {X 0,Y 337.333,Z 787.721,A -85,B 0,C 180,E1 -22161.787,E2 -22161.787} C_VEL
LIN {X 0,Y 337.908,Z 778.232,A -85,B 0,C 180,E1 -22162.871,E2 -22162.871} C_VEL
LIN {X 0,Y 338.512,Z 768.48,A -85,B 0,C 180,E1 -22163.796,E2 -22163.796} C_VEL
LIN {X 0,Y 339.035,Z 757.672,A -85,B 0,C 180,E1 -22164.627,E2 -22164.627} C_VEL
LIN {X 0,Y 339.369,Z 748.166,A -85,B 0,C 180,E1 -22165.214,E2 -22165.214} C_VEL
LIN {X 0,Y 339.804,Z 737.153,A -85,B 0,C 180,E1 -22165.732,E2 -22165.732} C_VEL
LIN {X 0,Y 340.615,Z 712.38,A -85,B 0,C 180,E1 -22166.527,E2 -22166.527} C_VEL
LIN {X 0,Y 342.01,Z 659.508,A -85,B 0,C 180,E1 -22168.125,E2 -22168.125} C_VEL
LIN {X 0,Y 339.136,Z 633.086,A -85,B 0,C 180,E1 -22169.002,E2 -22169.002} C_VEL
LIN {X 0,Y 338.755,Z 628.052,A -85,B 0,C 180,E1 -22169.167,E2 -22169.167} C_VEL
LIN {X 0,Y 339.248,Z 622.736,A -85,B 0,C 180,E1 -22170.73,E2 -22170.73} C_VEL
LIN {X 0,Y 337.992,Z 615.312,A -85,B 0,C 180,E1 -22173.044,E2 -22173.044} C_VEL
LIN {X 0,Y 337.783,Z 615.337,A -85,B 0,C 180,E1 -22176.967,E2 -22176.967} C_VEL
LIN {X 0,Y 337.77,Z 615.346,A -85,B 0,C 180,E1 -22180.004,E2 -22180.004} C_VEL
LIN {X 0,Y 337.809,Z 615.336,A -85,B 0,C 180,E1 -22183.471,E2 -22183.471} C_VEL
LIN {X 0,Y 337.806,Z 615.334,A -85,B 0,C 180,E1 -22186.822,E2 -22186.822} C_VEL
LIN {X 0,Y 337.77,Z 615.345,A -85,B 0,C 180,E1 -22190.109,E2 -22190.109} C_VEL
LIN {X 0,Y 337.809,Z 615.341,A -85,B 0,C 180,E1 -22193.964,E2 -22193.964} C_VEL
LIN {X 0,Y 337.778,Z 615.338,A -85,B 0,C 180,E1 -22197.373,E2 -22197.373} C_VEL
LIN {X 0,Y 337.82,Z 615.335,A -85,B 0,C 180,E1 -22200.555,E2 -22200.555} C_VEL
LIN {X 0,Y 337.823,Z 615.336,A -85,B 0,C 180,E1 -22204.188,E2 -22204.188} C_VEL
LIN {X 0,Y 337.825,Z 615.332,A -85,B 0,C 180,E1 -22206.8,E2 -22206.8} C_VEL
LIN {X 0,Y 337.896,Z 615.325,A -85,B 0,C 180,E1 -22209.365,E2 -22209.365} C_VEL
LIN {X 0,Y 337.933,Z 615.319,A -85,B 0,C 180,E1 -22213.131,E2 -22213.131} C_VEL
LIN {X 0,Y 338.026,Z 615.307,A -85,B 0,C 180,E1 -22216.882,E2 -22216.882} C_VEL
LIN {X 0,Y 338.046,Z 615.307,A -85,B 0,C 180,E1 -22220.458,E2 -22220.458} C_VEL
LIN {X 0,Y 338.204,Z 615.289,A -85,B 0,C 180,E1 -22224.056,E2 -22224.056} C_VEL
LIN {X 0,Y 338.238,Z 615.283,A -85,B 0,C 180,E1 -22227.626,E2 -22227.626} C_VEL
LIN {X 0,Y 338.206,Z 615.286,A -85,B 0,C 180,E1 -22231.186,E2 -22231.186} C_VEL
LIN {X 0,Y 338.245,Z 615.279,A -85,B 0,C 180,E1 -22234.751,E2 -22234.751} C_VEL
LIN {X 0,Y 338.086,Z 615.303,A -85,B 0,C 180,E1 -22238.339,E2 -22238.339} C_VEL
LIN {X 0,Y 338.004,Z 615.317,A -85,B 0,C 180,E1 -22241.96,E2 -22241.96} C_VEL
LIN {X 0,Y 337.932,Z 615.32,A -85,B 0,C 180,E1 -22244.402,E2 -22244.402} C_VEL
LIN {X 0,Y 337.88,Z 615.331,A -85,B 0,C 180,E1 -22248.117,E2 -22248.117} C_VEL
LIN {X 0,Y 337.88,Z 615.326,A -85,B 0,C 180,E1 -22251.114,E2 -22251.114} C_VEL
LIN {X 0,Y 337.836,Z 615.332,A -85,B 0,C 180,E1 -22254.498,E2 -22254.498} C_VEL
LIN {X 0,Y 337.839,Z 615.333,A -85,B 0,C 180,E1 -22258.48,E2 -22258.48} C_VEL
LIN {X 0,Y 337.804,Z 615.335,A -85,B 0,C 180,E1 -22262.623,E2 -22262.623} C_VEL
LIN {X 0,Y 337.875,Z 615.332,A -85,B 0,C 180,E1 -22266.051,E2 -22266.051} C_VEL
LIN {X 0,Y 337.84,Z 615.333,A -85,B 0,C 180,E1 -22268.461,E2 -22268.461} C_VEL
LIN {X 0,Y 337.814,Z 615.337,A -85,B 0,C 180,E1 -22271.718,E2 -22271.718} C_VEL
LIN {X 0,Y 337.807,Z 615.334,A -85,B 0,C 180,E1 -22275.172,E2 -22275.172} C_VEL
LIN {X 0,Y 337.821,Z 615.336,A -85,B 0,C 180,E1 -22278.434,E2 -22278.434} C_VEL
LIN {X 0,Y 337.816,Z 615.339,A -85,B 0,C 180,E1 -22281.99,E2 -22281.99} C_VEL
LIN {X 0,Y 337.814,Z 615.335,A -85,B 0,C 180,E1 -22284.51,E2 -22284.51} C_VEL
LIN {X 0,Y 337.813,Z 615.339,A -85,B 0,C 180,E1 -22288.225,E2 -22288.225} C_VEL
LIN {X 0,Y 337.84,Z 615.332,A -85,B 0,C 180,E1 -22291.52,E2 -22291.52} C_VEL
LIN {X 0,Y 337.838,Z 615.332,A -85,B 0,C 180,E1 -22295.502,E2 -22295.502} C_VEL
LIN {X 0,Y 337.897,Z 615.325,A -85,B 0,C 180,E1 -22299.366,E2 -22299.366} C_VEL
LIN {X 0,Y 337.911,Z 615.32,A -85,B 0,C 180,E1 -22303.131,E2 -22303.131} C_VEL
LIN {X 0,Y 338.026,Z 615.308,A -85,B 0,C 180,E1 -22306.884,E2 -22306.884} C_VEL
LIN {X 0,Y 338.049,Z 615.306,A -85,B 0,C 180,E1 -22310.459,E2 -22310.459} C_VEL
LIN {X 0,Y 338.244,Z 615.286,A -85,B 0,C 180,E1 -22314.057,E2 -22314.057} C_VEL
LIN {X 0,Y 338.242,Z 615.284,A -85,B 0,C 180,E1 -22317.627,E2 -22317.627} C_VEL
LIN {X 0,Y 338.207,Z 615.285,A -85,B 0,C 180,E1 -22321.187,E2 -22321.187} C_VEL
LIN {X 0,Y 338.244,Z 615.281,A -85,B 0,C 180,E1 -22324.752,E2 -22324.752} C_VEL
LIN {X 0,Y 338.159,Z 615.292,A -85,B 0,C 180,E1 -22327.14,E2 -22327.14} C_VEL
LIN {X 0,Y 337.99,Z 615.312,A -85,B 0,C 180,E1 -22330.75,E2 -22330.75} C_VEL
LIN {X 0,Y 337.978,Z 615.313,A -85,B 0,C 180,E1 -22333.178,E2 -22333.178} C_VEL
LIN {X 0,Y 337.872,Z 615.329,A -85,B 0,C 180,E1 -22337.517,E2 -22337.517} C_VEL
LIN {X 0,Y 337.841,Z 615.335,A -85,B 0,C 180,E1 -22338.223,E2 -22338.223} C_VEL
LIN {X 0,Y 337.125,Z 615.422,A -85,B 0,C 180,E1 -22339.218,E2 -22339.218} C_VEL
LIN {X 0,Y 334.225,Z 615.78,A -85,B 0,C 180,E1 -22340.836,E2 -22340.836} C_VEL
LIN {X 0,Y 331.821,Z 616.084,A -85,B 0,C 180,E1 -22342.147,E2 -22342.147} C_VEL
LIN {X 0,Y 330.831,Z 616.204,A -85,B 0,C 180,E1 -22343.161,E2 -22343.161} C_VEL
LIN {X 0,Y 330.772,Z 616.212,A -85,B 0,C 180,E1 -22343.505,E2 -22343.505} C_VEL
LIN {X 0,Y 330.788,Z 616.21,A -85,B 0,C 180,E1 -22347.209,E2 -22347.209} C_VEL
LIN {X 0,Y 330.721,Z 616.217,A -85,B 0,C 180,E1 -22350.551,E2 -22350.551} C_VEL
LIN {X 0,Y 330.747,Z 616.218,A -85,B 0,C 180,E1 -22354.318,E2 -22354.318} C_VEL
LIN {X 0,Y 330.74,Z 616.221,A -85,B 0,C 180,E1 -22357.892,E2 -22357.892} C_VEL
LIN {X 0,Y 330.701,Z 616.224,A -85,B 0,C 180,E1 -22362.156,E2 -22362.156} C_VEL
LIN {X 0,Y 330.693,Z 616.227,A -85,B 0,C 180,E1 -22366.068,E2 -22366.068} C_VEL
LIN {X 0,Y 330.688,Z 616.224,A -85,B 0,C 180,E1 -22369.688,E2 -22369.688} C_VEL
LIN {X 0,Y 330.725,Z 616.222,A -85,B 0,C 180,E1 -22372.107,E2 -22372.107} C_VEL
LIN {X 0,Y 330.738,Z 616.219,A -85,B 0,C 180,E1 -22375.685,E2 -22375.685} C_VEL
LIN {X 0,Y 330.71,Z 616.22,A -85,B 0,C 180,E1 -22379.448,E2 -22379.448} C_VEL
LIN {X 0,Y 330.852,Z 616.232,A -85,B 0,C 180,E1 -22383.037,E2 -22383.037} C_VEL
LIN {X 0,Y 332.941,Z 627.89,A -85,B 0,C 180,E1 -22386.439,E2 -22386.439} C_VEL
LIN {X 0,Y 332.858,Z 631.367,A -85,B 0,C 180,E1 -22387.416,E2 -22387.416} C_VEL
LIN {X 0,Y 331.357,Z 642.965,A -85,B 0,C 180,E1 -22390.63,E2 -22390.63} C_VEL
LIN {X 0,Y 332.519,Z 662.556,A -85,B 0,C 180,E1 -22391.303,E2 -22391.303} C_VEL
LIN {X 0,Y 334.62,Z 686.064,A -85,B 0,C 180,E1 -22392.095,E2 -22392.095} C_VEL
LIN {X 0,Y 332.851,Z 749.919,A -85,B 0,C 180,E1 -22394.123,E2 -22394.123} C_VEL
LIN {X 0,Y 332.385,Z 760.755,A -85,B 0,C 180,E1 -22394.61,E2 -22394.61} C_VEL
LIN {X 0,Y 332.017,Z 770.364,A -85,B 0,C 180,E1 -22395.179,E2 -22395.179} C_VEL
LIN {X 0,Y 331.539,Z 780.55,A -85,B 0,C 180,E1 -22395.939,E2 -22395.939} C_VEL
LIN {X 0,Y 331.009,Z 790.425,A -85,B 0,C 180,E1 -22396.847,E2 -22396.847} C_VEL
LIN {X 0,Y 330.368,Z 798.749,A -85,B 0,C 180,E1 -22397.759,E2 -22397.759} C_VEL
LIN {X 0,Y 329.884,Z 807.035,A -85,B 0,C 180,E1 -22398.828,E2 -22398.828} C_VEL
LIN {X 0,Y 329.347,Z 815.931,A -85,B 0,C 180,E1 -22400.204,E2 -22400.204} C_VEL
LIN {X 0,Y 328.904,Z 822.668,A -85,B 0,C 180,E1 -22401.427,E2 -22401.427} C_VEL
LIN {X 0,Y 328.664,Z 829.765,A -85,B 0,C 180,E1 -22402.961,E2 -22402.961} C_VEL
LIN {X 0,Y 328.464,Z 835.667,A -85,B 0,C 180,E1 -22404.494,E2 -22404.494} C_VEL
LIN {X 0,Y 328.338,Z 841.349,A -85,B 0,C 180,E1 -22406.331,E2 -22406.331} C_VEL
LIN {X 0,Y 328.304,Z 845.741,A -85,B 0,C 180,E1 -22408.166,E2 -22408.166} C_VEL
LIN {X 0,Y 328.203,Z 848.987,A -85,B 0,C 180,E1 -22410,E2 -22410} C_VEL
LIN {X 0,Y 328.12,Z 850.602,A -85,B 0,C 180,E1 -22411.223,E2 -22411.223} C_VEL
LIN {X 0,Y 328.065,Z 852.453,A -85,B 0,C 180,E1 -22413.673,E2 -22413.673} C_VEL
LIN {X 0,Y 328.152,Z 852.711,A -85,B 0,C 180,E1 -22414.898,E2 -22414.898} C_VEL
LIN {X 0,Y 328.693,Z 852.129,A -85,B 0,C 180,E1 -22417.346,E2 -22417.346} C_VEL
LIN {X 0,Y 329.739,Z 849.773,A -85,B 0,C 180,E1 -22419.785,E2 -22419.785} C_VEL
LIN {X 0,Y 330.956,Z 846.96,A -85,B 0,C 180,E1 -22421.599,E2 -22421.599} C_VEL
LIN {X 0,Y 332.651,Z 843.103,A -85,B 0,C 180,E1 -22423.393,E2 -22423.393} C_VEL
LIN {X 0,Y 334.64,Z 838.115,A -85,B 0,C 180,E1 -22425.168,E2 -22425.168} C_VEL
LIN {X 0,Y 336.9,Z 831.667,A -85,B 0,C 180,E1 -22426.985,E2 -22426.985} C_VEL
LIN {X 0,Y 339.11,Z 825.69,A -85,B 0,C 180,E1 -22428.361,E2 -22428.361} C_VEL
LIN {X 0,Y 341.54,Z 818.301,A -85,B 0,C 180,E1 -22429.779,E2 -22429.779} C_VEL
LIN {X 0,Y 344.19,Z 809.452,A -85,B 0,C 180,E1 -22431.175,E2 -22431.175} C_VEL
LIN {X 0,Y 346.568,Z 801.051,A -85,B 0,C 180,E1 -22432.269,E2 -22432.269} C_VEL
LIN {X 0,Y 349.114,Z 791.029,A -85,B 0,C 180,E1 -22433.344,E2 -22433.344} C_VEL
LIN {X 0,Y 351.218,Z 782.211,A -85,B 0,C 180,E1 -22434.132,E2 -22434.132} C_VEL
LIN {X 0,Y 353.412,Z 771.525,A -85,B 0,C 180,E1 -22434.908,E2 -22434.908} C_VEL
LIN {X 0,Y 355.342,Z 760.351,A -85,B 0,C 180,E1 -22435.544,E2 -22435.544} C_VEL
LIN {X 0,Y 356.804,Z 749.547,A -85,B 0,C 180,E1 -22436.017,E2 -22436.017} C_VEL
LIN {X 0,Y 361.626,Z 697.758,A -85,B 0,C 180,E1 -22437.702,E2 -22437.702} C_VEL
LIN {X 0,Y 359.898,Z 683.656,A -85,B 0,C 180,E1 -22438.715,E2 -22438.715} C_VEL
LIN {X 0,Y 358.549,Z 676.747,A -85,B 0,C 180,E1 -22439.327,E2 -22439.327} C_VEL
LIN {X 0,Y 354.532,Z 667.818,A -85,B 0,C 180,E1 -22440.618,E2 -22440.618} C_VEL
LIN {X 0,Y 350.82,Z 660.584,A -85,B 0,C 180,E1 -22441.861,E2 -22441.861} C_VEL
LIN {X 0,Y 348.094,Z 655.749,A -85,B 0,C 180,E1 -22442.818,E2 -22442.818} C_VEL
LIN {X 0,Y 345.04,Z 650.55,A -85,B 0,C 180,E1 -22443.976,E2 -22443.976} C_VEL
LIN {X 0,Y 342.124,Z 645.664,A -85,B 0,C 180,E1 -22445.18,E2 -22445.18} C_VEL
LIN {X 0,Y 338.231,Z 640.099,A -85,B 0,C 180,E1 -22446.911,E2 -22446.911} C_VEL
LIN {X 0,Y 337.639,Z 638.674,A -85,B 0,C 180,E1 -22447.327,E2 -22447.327} C_VEL
LIN {X 0,Y 336.616,Z 635.134,A -85,B 0,C 180,E1 -22450.171,E2 -22450.171} C_VEL
LIN {X 0,Y 335.724,Z 631.945,A -85,B 0,C 180,E1 -22453.512,E2 -22453.512} C_VEL
LIN {X 0,Y 335.102,Z 629.75,A -85,B 0,C 180,E1 -22457.02,E2 -22457.02} C_VEL
LIN {X 0,Y 334.884,Z 628.89,A -85,B 0,C 180,E1 -22459.579,E2 -22459.579} C_VEL
LIN {X 0,Y 334.773,Z 628.695,A -85,B 0,C 180,E1 -22462.662,E2 -22462.662} C_VEL
LIN {X 0,Y 334.977,Z 629.351,A -85,B 0,C 180,E1 -22465.627,E2 -22465.627} C_VEL
LIN {X 0,Y 335.473,Z 631.017,A -85,B 0,C 180,E1 -22468.877,E2 -22468.877} C_VEL
LIN {X 0,Y 336.212,Z 633.799,A -85,B 0,C 180,E1 -22472.257,E2 -22472.257} C_VEL
LIN {X 0,Y 338.6,Z 637.608,A -85,B 0,C 180,E1 -22473.527,E2 -22473.527} C_VEL
LIN {X 0,Y 340.728,Z 639.966,A -85,B 0,C 180,E1 -22474.44,E2 -22474.44} C_VEL
LIN {X 0,Y 343.398,Z 643.962,A -85,B 0,C 180,E1 -22475.607,E2 -22475.607} C_VEL
LIN {X 0,Y 344.914,Z 646.042,A -85,B 0,C 180,E1 -22476.192,E2 -22476.192} C_VEL
LIN {X 0,Y 348.09,Z 650.747,A -85,B 0,C 180,E1 -22477.366,E2 -22477.366} C_VEL
LIN {X 0,Y 351.369,Z 656.062,A -85,B 0,C 180,E1 -22478.505,E2 -22478.505} C_VEL
LIN {X 0,Y 355.374,Z 663.051,A -85,B 0,C 180,E1 -22479.808,E2 -22479.808} C_VEL
LIN {X 0,Y 360.363,Z 673.006,A -85,B 0,C 180,E1 -22481.327,E2 -22481.327} C_VEL
LIN {X 0,Y 363.057,Z 679.621,A -85,B 0,C 180,E1 -22482.162,E2 -22482.162} C_VEL
LIN {X 0,Y 357.231,Z 738.881,A -85,B 0,C 180,E1 -22484.067,E2 -22484.067} C_VEL
LIN {X 0,Y 355.901,Z 749.284,A -85,B 0,C 180,E1 -22484.533,E2 -22484.533} C_VEL
LIN {X 0,Y 354.339,Z 759.195,A -85,B 0,C 180,E1 -22485.109,E2 -22485.109} C_VEL
LIN {X 0,Y 352.331,Z 770.002,A -85,B 0,C 180,E1 -22485.905,E2 -22485.905} C_VEL
LIN {X 0,Y 350.127,Z 780.229,A -85,B 0,C 180,E1 -22486.846,E2 -22486.846} C_VEL
LIN {X 0,Y 347.198,Z 792.253,A -85,B 0,C 180,E1 -22488.213,E2 -22488.213} C_VEL
LIN {X 0,Y 344.187,Z 802.713,A -85,B 0,C 180,E1 -22489.742,E2 -22489.742} C_VEL
LIN {X 0,Y 341.652,Z 810.59,A -85,B 0,C 180,E1 -22491.155,E2 -22491.155} C_VEL
LIN {X 0,Y 339.281,Z 817.238,A -85,B 0,C 180,E1 -22492.594,E2 -22492.594} C_VEL
LIN {X 0,Y 337.132,Z 822.759,A -85,B 0,C 180,E1 -22494.037,E2 -22494.037} C_VEL
LIN {X 0,Y 334.835,Z 828.186,A -85,B 0,C 180,E1 -22495.801,E2 -22495.801} C_VEL
LIN {X 0,Y 332.884,Z 832.44,A -85,B 0,C 180,E1 -22497.588,E2 -22497.588} C_VEL
LIN {X 0,Y 331.801,Z 834.739,A -85,B 0,C 180,E1 -22498.79,E2 -22498.79} C_VEL
LIN {X 0,Y 330.112,Z 837.76,A -85,B 0,C 180,E1 -22501.215,E2 -22501.215} C_VEL
LIN {X 0,Y 329.524,Z 838.721,A -85,B 0,C 180,E1 -22502.498,E2 -22502.498} C_VEL
LIN {X 0,Y 328.547,Z 839.25,A -85,B 0,C 180,E1 -22504.892,E2 -22504.892} C_VEL
LIN {X 0,Y 328.217,Z 838.838,A -85,B 0,C 180,E1 -22506.125,E2 -22506.125} C_VEL
LIN {X 0,Y 327.886,Z 836.901,A -85,B 0,C 180,E1 -22508.6,E2 -22508.6} C_VEL
LIN {X 0,Y 327.899,Z 833.796,A -85,B 0,C 180,E1 -22510.692,E2 -22510.692} C_VEL
LIN {X 0,Y 327.892,Z 830.452,A -85,B 0,C 180,E1 -22512.334,E2 -22512.334} C_VEL
LIN {X 0,Y 328.173,Z 824.435,A -85,B 0,C 180,E1 -22514.524,E2 -22514.524} C_VEL
LIN {X 0,Y 328.455,Z 819.034,A -85,B 0,C 180,E1 -22516.094,E2 -22516.094} C_VEL
LIN {X 0,Y 328.788,Z 812.416,A -85,B 0,C 180,E1 -22517.672,E2 -22517.672} C_VEL
LIN {X 0,Y 329.216,Z 804.365,A -85,B 0,C 180,E1 -22519.255,E2 -22519.255} C_VEL
LIN {X 0,Y 329.663,Z 797.438,A -85,B 0,C 180,E1 -22520.416,E2 -22520.416} C_VEL
LIN {X 0,Y 330.246,Z 787.617,A -85,B 0,C 180,E1 -22521.787,E2 -22521.787} C_VEL
LIN {X 0,Y 330.821,Z 778.068,A -85,B 0,C 180,E1 -22522.895,E2 -22522.895} C_VEL
LIN {X 0,Y 331.434,Z 768.247,A -85,B 0,C 180,E1 -22523.839,E2 -22523.839} C_VEL
LIN {X 0,Y 331.909,Z 758.17,A -85,B 0,C 180,E1 -22524.632,E2 -22524.632} C_VEL
LIN {X 0,Y 332.293,Z 748.082,A -85,B 0,C 180,E1 -22525.267,E2 -22525.267} C_VEL
LIN {X 0,Y 332.747,Z 736.5,A -85,B 0,C 180,E1 -22525.815,E2 -22525.815} C_VEL
LIN {X 0,Y 333.814,Z 704.212,A -85,B 0,C 180,E1 -22526.858,E2 -22526.858} C_VEL
LIN {X 0,Y 334.906,Z 659.617,A -85,B 0,C 180,E1 -22528.26,E2 -22528.26} C_VEL
LIN {X 0,Y 332.07,Z 633.106,A -85,B 0,C 180,E1 -22529.163,E2 -22529.163} C_VEL
LIN {X 0,Y 331.731,Z 628.156,A -85,B 0,C 180,E1 -22529.349,E2 -22529.349} C_VEL
LIN {X 0,Y 332.188,Z 623.476,A -85,B 0,C 180,E1 -22530.752,E2 -22530.752} C_VEL
LIN {X 0,Y 330.945,Z 616.19,A -85,B 0,C 180,E1 -22533.091,E2 -22533.091} C_VEL
LIN {X 0,Y 330.749,Z 616.215,A -85,B 0,C 180,E1 -22536.414,E2 -22536.414} C_VEL
LIN {X 0,Y 330.718,Z 616.219,A -85,B 0,C 180,E1 -22539.448,E2 -22539.448} C_VEL
LIN {X 0,Y 330.733,Z 616.217,A -85,B 0,C 180,E1 -22542.664,E2 -22542.664} C_VEL
LIN {X 0,Y 330.755,Z 616.217,A -85,B 0,C 180,E1 -22546.055,E2 -22546.055} C_VEL
LIN {X 0,Y 330.71,Z 616.222,A -85,B 0,C 180,E1 -22549.682,E2 -22549.682} C_VEL
LIN {X 0,Y 330.741,Z 616.22,A -85,B 0,C 180,E1 -22552.109,E2 -22552.109} C_VEL
LIN {X 0,Y 330.749,Z 616.216,A -85,B 0,C 180,E1 -22555.681,E2 -22555.681} C_VEL
LIN {X 0,Y 330.748,Z 616.216,A -85,B 0,C 180,E1 -22559.451,E2 -22559.451} C_VEL
LIN {X 0,Y 330.786,Z 616.21,A -85,B 0,C 180,E1 -22562.791,E2 -22562.791} C_VEL
LIN {X 0,Y 330.788,Z 616.212,A -85,B 0,C 180,E1 -22566.276,E2 -22566.276} C_VEL
LIN {X 0,Y 330.85,Z 616.202,A -85,B 0,C 180,E1 -22568.905,E2 -22568.905} C_VEL
LIN {X 0,Y 330.907,Z 616.195,A -85,B 0,C 180,E1 -22572.762,E2 -22572.762} C_VEL
LIN {X 0,Y 330.977,Z 616.185,A -85,B 0,C 180,E1 -22576.776,E2 -22576.776} C_VEL
LIN {X 0,Y 330.992,Z 616.188,A -85,B 0,C 180,E1 -22580.253,E2 -22580.253} C_VEL
LIN {X 0,Y 331.19,Z 616.164,A -85,B 0,C 180,E1 -22583.93,E2 -22583.93} C_VEL
LIN {X 0,Y 331.204,Z 616.159,A -85,B 0,C 180,E1 -22587.576,E2 -22587.576} C_VEL
LIN {X 0,Y 331.183,Z 616.161,A -85,B 0,C 180,E1 -22591.212,E2 -22591.212} C_VEL
LIN {X 0,Y 331.19,Z 616.157,A -85,B 0,C 180,E1 -22594.853,E2 -22594.853} C_VEL
LIN {X 0,Y 331.107,Z 616.17,A -85,B 0,C 180,E1 -22597.292,E2 -22597.292} C_VEL
LIN {X 0,Y 330.934,Z 616.191,A -85,B 0,C 180,E1 -22600.981,E2 -22600.981} C_VEL
LIN {X 0,Y 330.974,Z 616.187,A -85,B 0,C 180,E1 -22603.461,E2 -22603.461} C_VEL
LIN {X 0,Y 330.865,Z 616.203,A -85,B 0,C 180,E1 -22607.704,E2 -22607.704} C_VEL
LIN {X 0,Y 330.82,Z 616.206,A -85,B 0,C 180,E1 -22611.315,E2 -22611.315} C_VEL
LIN {X 0,Y 330.788,Z 616.208,A -85,B 0,C 180,E1 -22615.056,E2 -22615.056} C_VEL
LIN {X 0,Y 330.775,Z 616.215,A -85,B 0,C 180,E1 -22617.766,E2 -22617.766} C_VEL
LIN {X 0,Y 330.749,Z 616.216,A -85,B 0,C 180,E1 -22620.548,E2 -22620.548} C_VEL
LIN {X 0,Y 330.79,Z 616.211,A -85,B 0,C 180,E1 -22624.329,E2 -22624.329} C_VEL
LIN {X 0,Y 330.803,Z 616.212,A -85,B 0,C 180,E1 -22627.882,E2 -22627.882} C_VEL
LIN {X 0,Y 330.751,Z 616.214,A -85,B 0,C 180,E1 -22631.033,E2 -22631.033} C_VEL
LIN {X 0,Y 330.752,Z 616.216,A -85,B 0,C 180,E1 -22634.335,E2 -22634.335} C_VEL
LIN {X 0,Y 330.744,Z 616.219,A -85,B 0,C 180,E1 -22637.836,E2 -22637.836} C_VEL
LIN {X 0,Y 330.783,Z 616.212,A -85,B 0,C 180,E1 -22641.581,E2 -22641.581} C_VEL
LIN {X 0,Y 330.753,Z 616.213,A -85,B 0,C 180,E1 -22645.126,E2 -22645.126} C_VEL
LIN {X 0,Y 330.765,Z 616.219,A -85,B 0,C 180,E1 -22648.035,E2 -22648.035} C_VEL
LIN {X 0,Y 330.772,Z 616.211,A -85,B 0,C 180,E1 -22650.854,E2 -22650.854} C_VEL
LIN {X 0,Y 330.765,Z 616.213,A -85,B 0,C 180,E1 -22653.596,E2 -22653.596} C_VEL
LIN {X 0,Y 330.79,Z 616.213,A -85,B 0,C 180,E1 -22656.277,E2 -22656.277} C_VEL
LIN {X 0,Y 330.852,Z 616.202,A -85,B 0,C 180,E1 -22658.906,E2 -22658.906} C_VEL
LIN {X 0,Y 330.872,Z 616.197,A -85,B 0,C 180,E1 -22662.76,E2 -22662.76} C_VEL
LIN {X 0,Y 330.958,Z 616.189,A -85,B 0,C 180,E1 -22666.793,E2 -22666.793} C_VEL
LIN {X 0,Y 330.994,Z 616.187,A -85,B 0,C 180,E1 -22670.254,E2 -22670.254} C_VEL
LIN {X 0,Y 331.221,Z 616.159,A -85,B 0,C 180,E1 -22673.931,E2 -22673.931} C_VEL
LIN {X 0,Y 331.207,Z 616.16,A -85,B 0,C 180,E1 -22677.576,E2 -22677.576} C_VEL
LIN {X 0,Y 331.184,Z 616.159,A -85,B 0,C 180,E1 -22681.212,E2 -22681.212} C_VEL
LIN {X 0,Y 331.19,Z 616.159,A -85,B 0,C 180,E1 -22684.853,E2 -22684.853} C_VEL
LIN {X 0,Y 331.111,Z 616.17,A -85,B 0,C 180,E1 -22687.292,E2 -22687.292} C_VEL
LIN {X 0,Y 330.935,Z 616.19,A -85,B 0,C 180,E1 -22690.982,E2 -22690.982} C_VEL
LIN {X 0,Y 330.906,Z 616.195,A -85,B 0,C 180,E1 -22693.465,E2 -22693.465} C_VEL
LIN {X 0,Y 330.818,Z 616.209,A -85,B 0,C 180,E1 -22697.676,E2 -22697.676} C_VEL
LIN {X 0,Y 330.776,Z 616.21,A -85,B 0,C 180,E1 -22701.293,E2 -22701.293} C_VEL
LIN {X 0,Y 330.772,Z 616.212,A -85,B 0,C 180,E1 -22703.505,E2 -22703.505} C_VEL
LIN {X 0,Y 330.158,Z 616.293,A -85,B 0,C 180,E1 -22704.522,E2 -22704.522} C_VEL
LIN {X 0,Y 327.309,Z 616.649,A -85,B 0,C 180,E1 -22706.177,E2 -22706.177} C_VEL
LIN {X 0,Y 324.853,Z 616.952,A -85,B 0,C 180,E1 -22707.518,E2 -22707.518} C_VEL
LIN {X 0,Y 323.786,Z 617.083,A -85,B 0,C 180,E1 -22708.556,E2 -22708.556} C_VEL
LIN {X 0,Y 323.694,Z 617.093,A -85,B 0,C 180,E1 -22708.908,E2 -22708.908} C_VEL
LIN {X 0,Y 323.687,Z 617.093,A -85,B 0,C 180,E1 -22712.751,E2 -22712.751} C_VEL
LIN {X 0,Y 323.704,Z 617.096,A -85,B 0,C 180,E1 -22715.749,E2 -22715.749} C_VEL
LIN {X 0,Y 323.697,Z 617.093,A -85,B 0,C 180,E1 -22718.868,E2 -22718.868} C_VEL
LIN {X 0,Y 323.665,Z 617.097,A -85,B 0,C 180,E1 -22722.626,E2 -22722.626} C_VEL
LIN {X 0,Y 323.661,Z 617.102,A -85,B 0,C 180,E1 -22726.17,E2 -22726.17} C_VEL
LIN {X 0,Y 323.643,Z 617.101,A -85,B 0,C 180,E1 -22729.513,E2 -22729.513} C_VEL
LIN {X 0,Y 323.67,Z 617.096,A -85,B 0,C 180,E1 -22732.704,E2 -22732.704} C_VEL
LIN {X 0,Y 323.689,Z 617.098,A -85,B 0,C 180,E1 -22735.763,E2 -22735.763} C_VEL
LIN {X 0,Y 323.642,Z 617.1,A -85,B 0,C 180,E1 -22738.707,E2 -22738.707} C_VEL
LIN {X 0,Y 323.824,Z 617.217,A -85,B 0,C 180,E1 -22743.028,E2 -22743.028} C_VEL
LIN {X 0,Y 325.951,Z 629.112,A -85,B 0,C 180,E1 -22746.575,E2 -22746.575} C_VEL
LIN {X 0,Y 325.154,Z 635.942,A -85,B 0,C 180,E1 -22748.518,E2 -22748.518} C_VEL
LIN {X 0,Y 324.313,Z 642.881,A -85,B 0,C 180,E1 -22750.483,E2 -22750.483} C_VEL
LIN {X 0,Y 325.607,Z 664.9,A -85,B 0,C 180,E1 -22751.256,E2 -22751.256} C_VEL
LIN {X 0,Y 327.532,Z 686.823,A -85,B 0,C 180,E1 -22752.013,E2 -22752.013} C_VEL
LIN {X 0,Y 325.755,Z 750.302,A -85,B 0,C 180,E1 -22754.089,E2 -22754.089} C_VEL
LIN {X 0,Y 325.31,Z 760.975,A -85,B 0,C 180,E1 -22754.587,E2 -22754.587} C_VEL
LIN {X 0,Y 324.93,Z 770.48,A -85,B 0,C 180,E1 -22755.168,E2 -22755.168} C_VEL
LIN {X 0,Y 324.455,Z 780.605,A -85,B 0,C 180,E1 -22755.944,E2 -22755.944} C_VEL
LIN {X 0,Y 323.902,Z 790.388,A -85,B 0,C 180,E1 -22756.867,E2 -22756.867} C_VEL
LIN {X 0,Y 323.255,Z 798.723,A -85,B 0,C 180,E1 -22757.804,E2 -22757.804} C_VEL
LIN {X 0,Y 322.776,Z 806.99,A -85,B 0,C 180,E1 -22758.896,E2 -22758.896} C_VEL
LIN {X 0,Y 322.234,Z 815.87,A -85,B 0,C 180,E1 -22760.302,E2 -22760.302} C_VEL
LIN {X 0,Y 321.827,Z 822.59,A -85,B 0,C 180,E1 -22761.552,E2 -22761.552} C_VEL
LIN {X 0,Y 321.586,Z 829.637,A -85,B 0,C 180,E1 -22763.12,E2 -22763.12} C_VEL
LIN {X 0,Y 321.39,Z 835.499,A -85,B 0,C 180,E1 -22764.686,E2 -22764.686} C_VEL
LIN {X 0,Y 321.301,Z 840.357,A -85,B 0,C 180,E1 -22766.25,E2 -22766.25} C_VEL
LIN {X 0,Y 321.239,Z 844.948,A -85,B 0,C 180,E1 -22768.126,E2 -22768.126} C_VEL
LIN {X 0,Y 321.128,Z 848.377,A -85,B 0,C 180,E1 -22770,E2 -22770} C_VEL
LIN {X 0,Y 321.025,Z 851.237,A -85,B 0,C 180,E1 -22772.501,E2 -22772.501} C_VEL
LIN {X 0,Y 320.976,Z 852.145,A -85,B 0,C 180,E1 -22773.754,E2 -22773.754} C_VEL
LIN {X 0,Y 321.306,Z 852.481,A -85,B 0,C 180,E1 -22776.258,E2 -22776.258} C_VEL
LIN {X 0,Y 321.63,Z 852.07,A -85,B 0,C 180,E1 -22777.508,E2 -22777.508} C_VEL
LIN {X 0,Y 322.761,Z 850.053,A -85,B 0,C 180,E1 -22779.998,E2 -22779.998} C_VEL
LIN {X 0,Y 324.023,Z 847.408,A -85,B 0,C 180,E1 -22781.851,E2 -22781.851} C_VEL
LIN {X 0,Y 325.802,Z 843.73,A -85,B 0,C 180,E1 -22783.68,E2 -22783.68} C_VEL
LIN {X 0,Y 327.867,Z 839.01,A -85,B 0,C 180,E1 -22785.489,E2 -22785.489} C_VEL
LIN {X 0,Y 330.337,Z 832.59,A -85,B 0,C 180,E1 -22787.412,E2 -22787.412} C_VEL
LIN {X 0,Y 333.019,Z 825.739,A -85,B 0,C 180,E1 -22789.027,E2 -22789.027} C_VEL
LIN {X 0,Y 335.565,Z 818.378,A -85,B 0,C 180,E1 -22790.465,E2 -22790.465} C_VEL
LIN {X 0,Y 338.353,Z 809.592,A -85,B 0,C 180,E1 -22791.878,E2 -22791.878} C_VEL
LIN {X 0,Y 341.19,Z 800.194,A -85,B 0,C 180,E1 -22793.118,E2 -22793.118} C_VEL
LIN {X 0,Y 343.536,Z 791.577,A -85,B 0,C 180,E1 -22794.066,E2 -22794.066} C_VEL
LIN {X 0,Y 346.076,Z 781.222,A -85,B 0,C 180,E1 -22794.993,E2 -22794.993} C_VEL
LIN {X 0,Y 348.188,Z 771.362,A -85,B 0,C 180,E1 -22795.707,E2 -22795.707} C_VEL
LIN {X 0,Y 350.199,Z 760.194,A -85,B 0,C 180,E1 -22796.346,E2 -22796.346} C_VEL
LIN {X 0,Y 351.733,Z 749.413,A -85,B 0,C 180,E1 -22796.82,E2 -22796.82} C_VEL
LIN {X 0,Y 356.699,Z 698.956,A -85,B 0,C 180,E1 -22798.521,E2 -22798.521} C_VEL
LIN {X 0,Y 355.206,Z 686.309,A -85,B 0,C 180,E1 -22799.457,E2 -22799.457} C_VEL
LIN {X 0,Y 354.104,Z 680.633,A -85,B 0,C 180,E1 -22799.976,E2 -22799.976} C_VEL
LIN {X 0,Y 349.898,Z 670.948,A -85,B 0,C 180,E1 -22801.453,E2 -22801.453} C_VEL
LIN {X 0,Y 346.296,Z 664.073,A -85,B 0,C 180,E1 -22802.736,E2 -22802.736} C_VEL
LIN {X 0,Y 344.66,Z 661.094,A -85,B 0,C 180,E1 -22803.363,E2 -22803.363} C_VEL
LIN {X 0,Y 341.83,Z 656.189,A -85,B 0,C 180,E1 -22804.477,E2 -22804.477} C_VEL
LIN {X 0,Y 338.662,Z 650.789,A -85,B 0,C 180,E1 -22805.885,E2 -22805.885} C_VEL
LIN {X 0,Y 335.586,Z 646.15,A -85,B 0,C 180,E1 -22807.346,E2 -22807.346} C_VEL
LIN {X 0,Y 334.635,Z 644.548,A -85,B 0,C 180,E1 -22807.862,E2 -22807.862} C_VEL
LIN {X 0,Y 331.023,Z 639.657,A -85,B 0,C 180,E1 -22809.947,E2 -22809.947} C_VEL
LIN {X 0,Y 330.263,Z 638.097,A -85,B 0,C 180,E1 -22810.563,E2 -22810.563} C_VEL
LIN {X 0,Y 329.467,Z 635.248,A -85,B 0,C 180,E1 -22813.711,E2 -22813.711} C_VEL
LIN {X 0,Y 328.938,Z 633.226,A -85,B 0,C 180,E1 -22817.046,E2 -22817.046} C_VEL
LIN {X 0,Y 328.657,Z 632.304,A -85,B 0,C 180,E1 -22820.108,E2 -22820.108} C_VEL
LIN {X 0,Y 328.591,Z 632.304,A -85,B 0,C 180,E1 -22823.354,E2 -22823.354} C_VEL
LIN {X 0,Y 328.856,Z 633.128,A -85,B 0,C 180,E1 -22826.373,E2 -22826.373} C_VEL
LIN {X 0,Y 329.336,Z 634.647,A -85,B 0,C 180,E1 -22829.043,E2 -22829.043} C_VEL
LIN {X 0,Y 332.24,Z 638.803,A -85,B 0,C 180,E1 -22831.059,E2 -22831.059} C_VEL
LIN {X 0,Y 334.057,Z 640.693,A -85,B 0,C 180,E1 -22832.048,E2 -22832.048} C_VEL
LIN {X 0,Y 337.003,Z 644.938,A -85,B 0,C 180,E1 -22833.593,E2 -22833.593} C_VEL
LIN {X 0,Y 338.324,Z 646.682,A -85,B 0,C 180,E1 -22834.188,E2 -22834.188} C_VEL
LIN {X 0,Y 341.266,Z 650.806,A -85,B 0,C 180,E1 -22835.475,E2 -22835.475} C_VEL
LIN {X 0,Y 345.139,Z 656.862,A -85,B 0,C 180,E1 -22836.994,E2 -22836.994} C_VEL
LIN {X 0,Y 348.179,Z 662.014,A -85,B 0,C 180,E1 -22838.124,E2 -22838.124} C_VEL
LIN {X 0,Y 352.226,Z 669.377,A -85,B 0,C 180,E1 -22839.49,E2 -22839.49} C_VEL
LIN {X 0,Y 356.204,Z 677.669,A -85,B 0,C 180,E1 -22840.786,E2 -22840.786} C_VEL
LIN {X 0,Y 358.08,Z 682.071,A -85,B 0,C 180,E1 -22841.372,E2 -22841.372} C_VEL
LIN {X 0,Y 352.135,Z 739.289,A -85,B 0,C 180,E1 -22843.273,E2 -22843.273} C_VEL
LIN {X 0,Y 350.473,Z 751.323,A -85,B 0,C 180,E1 -22843.825,E2 -22843.825} C_VEL
LIN {X 0,Y 348.205,Z 764.747,A -85,B 0,C 180,E1 -22844.676,E2 -22844.676} C_VEL
LIN {X 0,Y 345.795,Z 776.088,A -85,B 0,C 180,E1 -22845.632,E2 -22845.632} C_VEL
LIN {X 0,Y 343.194,Z 786.513,A -85,B 0,C 180,E1 -22846.726,E2 -22846.726} C_VEL
LIN {X 0,Y 340.777,Z 795.209,A -85,B 0,C 180,E1 -22847.837,E2 -22847.837} C_VEL
LIN {X 0,Y 338.506,Z 802.639,A -85,B 0,C 180,E1 -22848.965,E2 -22848.965} C_VEL
LIN {X 0,Y 335.822,Z 810.562,A -85,B 0,C 180,E1 -22850.394,E2 -22850.394} C_VEL
LIN {X 0,Y 333.223,Z 817.361,A -85,B 0,C 180,E1 -22851.871,E2 -22851.871} C_VEL
LIN {X 0,Y 331.023,Z 822.836,A -85,B 0,C 180,E1 -22853.316,E2 -22853.316} C_VEL
LIN {X 0,Y 328.546,Z 828.27,A -85,B 0,C 180,E1 -22855.108,E2 -22855.108} C_VEL
LIN {X 0,Y 326.413,Z 832.523,A -85,B 0,C 180,E1 -22856.924,E2 -22856.924} C_VEL
LIN {X 0,Y 324.7,Z 835.723,A -85,B 0,C 180,E1 -22858.764,E2 -22858.764} C_VEL
LIN {X 0,Y 323.814,Z 837.319,A -85,B 0,C 180,E1 -22860,E2 -22860} C_VEL
LIN {X 0,Y 322.426,Z 839.155,A -85,B 0,C 180,E1 -22862.49,E2 -22862.49} C_VEL
LIN {X 0,Y 321.506,Z 839.297,A -85,B 0,C 180,E1 -22864.719,E2 -22864.719} C_VEL
LIN {X 0,Y 321.091,Z 838.816,A -85,B 0,C 180,E1 -22866.261,E2 -22866.261} C_VEL
LIN {X 0,Y 320.782,Z 836.353,A -85,B 0,C 180,E1 -22868.792,E2 -22868.792} C_VEL
LIN {X 0,Y 320.821,Z 833.292,A -85,B 0,C 180,E1 -22870.74,E2 -22870.74} C_VEL
LIN {X 0,Y 320.836,Z 829.257,A -85,B 0,C 180,E1 -22872.61,E2 -22872.61} C_VEL
LIN {X 0,Y 321.034,Z 824.91,A -85,B 0,C 180,E1 -22874.208,E2 -22874.208} C_VEL
LIN {X 0,Y 321.337,Z 819.586,A -85,B 0,C 180,E1 -22875.811,E2 -22875.811} C_VEL
LIN {X 0,Y 321.656,Z 813.24,A -85,B 0,C 180,E1 -22877.39,E2 -22877.39} C_VEL
LIN {X 0,Y 322.057,Z 805.175,A -85,B 0,C 180,E1 -22879.04,E2 -22879.04} C_VEL
LIN {X 0,Y 322.62,Z 796.318,A -85,B 0,C 180,E1 -22880.542,E2 -22880.542} C_VEL
LIN {X 0,Y 323.146,Z 787.501,A -85,B 0,C 180,E1 -22881.789,E2 -22881.789} C_VEL
LIN {X 0,Y 323.722,Z 777.893,A -85,B 0,C 180,E1 -22882.921,E2 -22882.921} C_VEL
LIN {X 0,Y 324.352,Z 768.011,A -85,B 0,C 180,E1 -22883.885,E2 -22883.885} C_VEL
LIN {X 0,Y 324.792,Z 758.798,A -85,B 0,C 180,E1 -22884.628,E2 -22884.628} C_VEL
LIN {X 0,Y 325.222,Z 748.05,A -85,B 0,C 180,E1 -22885.321,E2 -22885.321} C_VEL
LIN {X 0,Y 325.658,Z 736.894,A -85,B 0,C 180,E1 -22885.862,E2 -22885.862} C_VEL
LIN {X 0,Y 326.598,Z 708.541,A -85,B 0,C 180,E1 -22886.811,E2 -22886.811} C_VEL
LIN {X 0,Y 327.909,Z 660.636,A -85,B 0,C 180,E1 -22888.352,E2 -22888.352} C_VEL
LIN {X 0,Y 325.175,Z 635.271,A -85,B 0,C 180,E1 -22889.243,E2 -22889.243} C_VEL
LIN {X 0,Y 324.697,Z 628.301,A -85,B 0,C 180,E1 -22889.505,E2 -22889.505} C_VEL
LIN {X 0,Y 325.126,Z 624.262,A -85,B 0,C 180,E1 -22890.743,E2 -22890.743} C_VEL
LIN {X 0,Y 323.896,Z 617.068,A -85,B 0,C 180,E1 -22893.095,E2 -22893.095} C_VEL
LIN {X 0,Y 323.685,Z 617.093,A -85,B 0,C 180,E1 -22897.294,E2 -22897.294} C_VEL
LIN {X 0,Y 323.693,Z 617.094,A -85,B 0,C 180,E1 -22900.767,E2 -22900.767} C_VEL
LIN {X 0,Y 323.705,Z 617.093,A -85,B 0,C 180,E1 -22904.433,E2 -22904.433} C_VEL
LIN {X 0,Y 323.684,Z 617.097,A -85,B 0,C 180,E1 -22907.868,E2 -22907.868} C_VEL
LIN {X 0,Y 323.7,Z 617.093,A -85,B 0,C 180,E1 -22911.167,E2 -22911.167} C_VEL
LIN {X 0,Y 323.723,Z 617.089,A -85,B 0,C 180,E1 -22915.306,E2 -22915.306} C_VEL
LIN {X 0,Y 323.684,Z 617.095,A -85,B 0,C 180,E1 -22918.711,E2 -22918.711} C_VEL
LIN {X 0,Y 323.732,Z 617.09,A -85,B 0,C 180,E1 -22922.509,E2 -22922.509} C_VEL
LIN {X 0,Y 323.765,Z 617.086,A -85,B 0,C 180,E1 -22925.729,E2 -22925.729} C_VEL
LIN {X 0,Y 323.776,Z 617.087,A -85,B 0,C 180,E1 -22929.748,E2 -22929.748} C_VEL
LIN {X 0,Y 323.82,Z 617.08,A -85,B 0,C 180,E1 -22933.668,E2 -22933.668} C_VEL
LIN {X 0,Y 323.936,Z 617.064,A -85,B 0,C 180,E1 -22937.512,E2 -22937.512} C_VEL
LIN {X 0,Y 323.995,Z 617.057,A -85,B 0,C 180,E1 -22941.296,E2 -22941.296} C_VEL
LIN {X 0,Y 324.146,Z 617.04,A -85,B 0,C 180,E1 -22943.797,E2 -22943.797} C_VEL
LIN {X 0,Y 324.155,Z 617.037,A -85,B 0,C 180,E1 -22947.523,E2 -22947.523} C_VEL
LIN {X 0,Y 324.161,Z 617.036,A -85,B 0,C 180,E1 -22951.238,E2 -22951.238} C_VEL
LIN {X 0,Y 324.139,Z 617.035,A -85,B 0,C 180,E1 -22954.958,E2 -22954.958} C_VEL
LIN {X 0,Y 324.053,Z 617.049,A -85,B 0,C 180,E1 -22957.451,E2 -22957.451} C_VEL
LIN {X 0,Y 323.883,Z 617.07,A -85,B 0,C 180,E1 -22961.223,E2 -22961.223} C_VEL
LIN {X 0,Y 323.912,Z 617.069,A -85,B 0,C 180,E1 -22963.761,E2 -22963.761} C_VEL
LIN {X 0,Y 323.815,Z 617.082,A -85,B 0,C 180,E1 -22967.871,E2 -22967.871} C_VEL
LIN {X 0,Y 323.772,Z 617.086,A -85,B 0,C 180,E1 -22971.578,E2 -22971.578} C_VEL
LIN {X 0,Y 323.751,Z 617.085,A -85,B 0,C 180,E1 -22974.678,E2 -22974.678} C_VEL
LIN {X 0,Y 323.717,Z 617.093,A -85,B 0,C 180,E1 -22978.426,E2 -22978.426} C_VEL
LIN {X 0,Y 323.723,Z 617.09,A -85,B 0,C 180,E1 -22982.453,E2 -22982.453} C_VEL
LIN {X 0,Y 323.755,Z 617.087,A -85,B 0,C 180,E1 -22985.742,E2 -22985.742} C_VEL
LIN {X 0,Y 323.75,Z 617.087,A -85,B 0,C 180,E1 -22988.86,E2 -22988.86} C_VEL
LIN {X 0,Y 323.705,Z 617.091,A -85,B 0,C 180,E1 -22992.634,E2 -22992.634} C_VEL
LIN {X 0,Y 323.714,Z 617.095,A -85,B 0,C 180,E1 -22996.18,E2 -22996.18} C_VEL
LIN {X 0,Y 323.697,Z 617.095,A -85,B 0,C 180,E1 -22999.522,E2 -22999.522} C_VEL
LIN {X 0,Y 323.73,Z 617.087,A -85,B 0,C 180,E1 -23003.183,E2 -23003.183} C_VEL
LIN {X 0,Y 323.704,Z 617.095,A -85,B 0,C 180,E1 -23005.765,E2 -23005.765} C_VEL
LIN {X 0,Y 323.686,Z 617.095,A -85,B 0,C 180,E1 -23008.712,E2 -23008.712} C_VEL
LIN {X 0,Y 323.733,Z 617.088,A -85,B 0,C 180,E1 -23012.51,E2 -23012.51} C_VEL
LIN {X 0,Y 323.766,Z 617.087,A -85,B 0,C 180,E1 -23015.73,E2 -23015.73} C_VEL
LIN {X 0,Y 323.777,Z 617.087,A -85,B 0,C 180,E1 -23019.749,E2 -23019.749} C_VEL
LIN {X 0,Y 323.814,Z 617.078,A -85,B 0,C 180,E1 -23022.373,E2 -23022.373} C_VEL
LIN {X 0,Y 323.902,Z 617.068,A -85,B 0,C 180,E1 -23026.688,E2 -23026.688} C_VEL
LIN {X 0,Y 324.003,Z 617.054,A -85,B 0,C 180,E1 -23031.296,E2 -23031.296} C_VEL
LIN {X 0,Y 324.189,Z 617.033,A -85,B 0,C 180,E1 -23033.799,E2 -23033.799} C_VEL
LIN {X 0,Y 324.159,Z 617.037,A -85,B 0,C 180,E1 -23037.524,E2 -23037.524} C_VEL
LIN {X 0,Y 324.162,Z 617.034,A -85,B 0,C 180,E1 -23041.239,E2 -23041.239} C_VEL
LIN {X 0,Y 324.14,Z 617.037,A -85,B 0,C 180,E1 -23044.959,E2 -23044.959} C_VEL
LIN {X 0,Y 324.057,Z 617.05,A -85,B 0,C 180,E1 -23047.452,E2 -23047.452} C_VEL
LIN {X 0,Y 323.882,Z 617.069,A -85,B 0,C 180,E1 -23051.224,E2 -23051.224} C_VEL
LIN {X 0,Y 323.835,Z 617.078,A -85,B 0,C 180,E1 -23053.764,E2 -23053.764} C_VEL
LIN {X 0,Y 323.776,Z 617.088,A -85,B 0,C 180,E1 -23057.847,E2 -23057.847} C_VEL
LIN {X 0,Y 323.714,Z 617.091,A -85,B 0,C 180,E1 -23061.583,E2 -23061.583} C_VEL
LIN {X 0,Y 323.755,Z 617.086,A -85,B 0,C 180,E1 -23064.678,E2 -23064.678} C_VEL
LIN {X 0,Y 323.719,Z 617.092,A -85,B 0,C 180,E1 -23068.426,E2 -23068.426} C_VEL
LIN {X 0,Y 323.694,Z 617.093,A -85,B 0,C 180,E1 -23068.908,E2 -23068.908} C_VEL
LIN {X 0,Y 323.005,Z 617.184,A -85,B 0,C 180,E1 -23069.947,E2 -23069.947} C_VEL
LIN {X 0,Y 320.121,Z 617.539,A -85,B 0,C 180,E1 -23071.637,E2 -23071.637} C_VEL
LIN {X 0,Y 317.702,Z 617.838,A -85,B 0,C 180,E1 -23073.007,E2 -23073.007} C_VEL
LIN {X 0,Y 316.688,Z 617.971,A -85,B 0,C 180,E1 -23074.068,E2 -23074.068} C_VEL
LIN {X 0,Y 316.617,Z 617.972,A -85,B 0,C 180,E1 -23074.427,E2 -23074.427} C_VEL
LIN {X 0,Y 316.641,Z 617.975,A -85,B 0,C 180,E1 -23078.272,E2 -23078.272} C_VEL
LIN {X 0,Y 316.596,Z 617.977,A -85,B 0,C 180,E1 -23081.585,E2 -23081.585} C_VEL
LIN {X 0,Y 316.608,Z 617.976,A -85,B 0,C 180,E1 -23085.069,E2 -23085.069} C_VEL
LIN {X 0,Y 316.602,Z 617.976,A -85,B 0,C 180,E1 -23088.782,E2 -23088.782} C_VEL
LIN {X 0,Y 316.641,Z 617.971,A -85,B 0,C 180,E1 -23092.784,E2 -23092.784} C_VEL
LIN {X 0,Y 316.616,Z 617.977,A -85,B 0,C 180,E1 -23096.422,E2 -23096.422} C_VEL
LIN {X 0,Y 316.622,Z 617.976,A -85,B 0,C 180,E1 -23099.63,E2 -23099.63} C_VEL
LIN {X 0,Y 316.793,Z 618.076,A -85,B 0,C 180,E1 -23103.002,E2 -23103.002} C_VEL
LIN {X 0,Y 318.788,Z 629.11,A -85,B 0,C 180,E1 -23106.36,E2 -23106.36} C_VEL
LIN {X 0,Y 318.523,Z 633.248,A -85,B 0,C 180,E1 -23107.571,E2 -23107.571} C_VEL
LIN {X 0,Y 317.263,Z 642.738,A -85,B 0,C 180,E1 -23110.325,E2 -23110.325} C_VEL
LIN {X 0,Y 318.4,Z 663.473,A -85,B 0,C 180,E1 -23111.077,E2 -23111.077} C_VEL
LIN {X 0,Y 320.488,Z 687.075,A -85,B 0,C 180,E1 -23111.912,E2 -23111.912} C_VEL
LIN {X 0,Y 318.691,Z 749.68,A -85,B 0,C 180,E1 -23114.013,E2 -23114.013} C_VEL
LIN {X 0,Y 318.215,Z 760.432,A -85,B 0,C 180,E1 -23114.521,E2 -23114.521} C_VEL
LIN {X 0,Y 317.82,Z 770.573,A -85,B 0,C 180,E1 -23115.155,E2 -23115.155} C_VEL
LIN {X 0,Y 317.45,Z 778.851,A -85,B 0,C 180,E1 -23115.791,E2 -23115.791} C_VEL
LIN {X 0,Y 316.863,Z 789.387,A -85,B 0,C 180,E1 -23116.791,E2 -23116.791} C_VEL
LIN {X 0,Y 316.153,Z 798.586,A -85,B 0,C 180,E1 -23117.85,E2 -23117.85} C_VEL
LIN {X 0,Y 315.698,Z 806.814,A -85,B 0,C 180,E1 -23118.968,E2 -23118.968} C_VEL
LIN {X 0,Y 315.163,Z 815.65,A -85,B 0,C 180,E1 -23120.405,E2 -23120.405} C_VEL
LIN {X 0,Y 314.738,Z 822.347,A -85,B 0,C 180,E1 -23121.683,E2 -23121.683} C_VEL
LIN {X 0,Y 314.514,Z 829.41,A -85,B 0,C 180,E1 -23123.286,E2 -23123.286} C_VEL
LIN {X 0,Y 314.326,Z 835.283,A -85,B 0,C 180,E1 -23124.886,E2 -23124.886} C_VEL
LIN {X 0,Y 314.204,Z 840.936,A -85,B 0,C 180,E1 -23126.805,E2 -23126.805} C_VEL
LIN {X 0,Y 314.164,Z 845.333,A -85,B 0,C 180,E1 -23128.723,E2 -23128.723} C_VEL
LIN {X 0,Y 314.063,Z 847.667,A -85,B 0,C 180,E1 -23130,E2 -23130} C_VEL
LIN {X 0,Y 313.943,Z 850.8,A -85,B 0,C 180,E1 -23132.558,E2 -23132.558} C_VEL
LIN {X 0,Y 313.899,Z 851.71,A -85,B 0,C 180,E1 -23133.839,E2 -23133.839} C_VEL
LIN {X 0,Y 314.24,Z 852.381,A -85,B 0,C 180,E1 -23136.399,E2 -23136.399} C_VEL
LIN {X 0,Y 315.053,Z 851.299,A -85,B 0,C 180,E1 -23138.953,E2 -23138.953} C_VEL
LIN {X 0,Y 315.762,Z 850.221,A -85,B 0,C 180,E1 -23140.222,E2 -23140.222} C_VEL
LIN {X 0,Y 317.677,Z 846.719,A -85,B 0,C 180,E1 -23142.738,E2 -23142.738} C_VEL
LIN {X 0,Y 319.602,Z 842.951,A -85,B 0,C 180,E1 -23144.598,E2 -23144.598} C_VEL
LIN {X 0,Y 321.894,Z 838.067,A -85,B 0,C 180,E1 -23146.433,E2 -23146.433} C_VEL
LIN {X 0,Y 324.258,Z 832.207,A -85,B 0,C 180,E1 -23148.189,E2 -23148.189} C_VEL
LIN {X 0,Y 327.46,Z 824.401,A -85,B 0,C 180,E1 -23150.014,E2 -23150.014} C_VEL
LIN {X 0,Y 330.178,Z 816.938,A -85,B 0,C 180,E1 -23151.466,E2 -23151.466} C_VEL
LIN {X 0,Y 332.588,Z 809.969,A -85,B 0,C 180,E1 -23152.604,E2 -23152.604} C_VEL
LIN {X 0,Y 335.579,Z 800.638,A -85,B 0,C 180,E1 -23153.854,E2 -23153.854} C_VEL
LIN {X 0,Y 338.349,Z 790.743,A -85,B 0,C 180,E1 -23154.949,E2 -23154.949} C_VEL
LIN {X 0,Y 341.031,Z 780.22,A -85,B 0,C 180,E1 -23155.878,E2 -23155.878} C_VEL
LIN {X 0,Y 343.473,Z 769.297,A -85,B 0,C 180,E1 -23156.657,E2 -23156.657} C_VEL
LIN {X 0,Y 345.347,Z 759.17,A -85,B 0,C 180,E1 -23157.234,E2 -23157.234} C_VEL
LIN {X 0,Y 346.867,Z 749.181,A -85,B 0,C 180,E1 -23157.675,E2 -23157.675} C_VEL
LIN {X 0,Y 351.912,Z 700.652,A -85,B 0,C 180,E1 -23159.326,E2 -23159.326} C_VEL
LIN {X 0,Y 350.493,Z 688.043,A -85,B 0,C 180,E1 -23160.312,E2 -23160.312} C_VEL
LIN {X 0,Y 349.881,Z 684.768,A -85,B 0,C 180,E1 -23160.633,E2 -23160.633} C_VEL
LIN {X 0,Y 346.162,Z 676.006,A -85,B 0,C 180,E1 -23161.998,E2 -23161.998} C_VEL
LIN {X 0,Y 342.16,Z 667.815,A -85,B 0,C 180,E1 -23163.576,E2 -23163.576} C_VEL
LIN {X 0,Y 338.639,Z 661.735,A -85,B 0,C 180,E1 -23165.022,E2 -23165.022} C_VEL
LIN {X 0,Y 335.829,Z 656.785,A -85,B 0,C 180,E1 -23166.338,E2 -23166.338} C_VEL
LIN {X 0,Y 332.945,Z 652.15,A -85,B 0,C 180,E1 -23167.807,E2 -23167.807} C_VEL
LIN {X 0,Y 332.031,Z 650.686,A -85,B 0,C 180,E1 -23168.325,E2 -23168.325} C_VEL
LIN {X 0,Y 328.706,Z 645.895,A -85,B 0,C 180,E1 -23170.374,E2 -23170.374} C_VEL
LIN {X 0,Y 327.856,Z 644.429,A -85,B 0,C 180,E1 -23171.018,E2 -23171.018} C_VEL
LIN {X 0,Y 323.531,Z 638.514,A -85,B 0,C 180,E1 -23175.173,E2 -23175.173} C_VEL
LIN {X 0,Y 322.801,Z 636.991,A -85,B 0,C 180,E1 -23176.496,E2 -23176.496} C_VEL
LIN {X 0,Y 322.545,Z 635.942,A -85,B 0,C 180,E1 -23179.471,E2 -23179.471} C_VEL
LIN {X 0,Y 322.421,Z 635.789,A -85,B 0,C 180,E1 -23182.982,E2 -23182.982} C_VEL
LIN {X 0,Y 324.126,Z 638.31,A -85,B 0,C 180,E1 -23185.928,E2 -23185.928} C_VEL
LIN {X 0,Y 327.391,Z 641.497,A -85,B 0,C 180,E1 -23188.848,E2 -23188.848} C_VEL
LIN {X 0,Y 330.375,Z 645.67,A -85,B 0,C 180,E1 -23190.957,E2 -23190.957} C_VEL
LIN {X 0,Y 331.695,Z 647.116,A -85,B 0,C 180,E1 -23191.697,E2 -23191.697} C_VEL
LIN {X 0,Y 334.754,Z 651.532,A -85,B 0,C 180,E1 -23193.366,E2 -23193.366} C_VEL
LIN {X 0,Y 339.205,Z 658.191,A -85,B 0,C 180,E1 -23195.402,E2 -23195.402} C_VEL
LIN {X 0,Y 342.222,Z 663.045,A -85,B 0,C 180,E1 -23196.63,E2 -23196.63} C_VEL
LIN {X 0,Y 344.85,Z 667.586,A -85,B 0,C 180,E1 -23197.649,E2 -23197.649} C_VEL
LIN {X 0,Y 348.641,Z 674.744,A -85,B 0,C 180,E1 -23199.008,E2 -23199.008} C_VEL
LIN {X 0,Y 352.597,Z 683.492,A -85,B 0,C 180,E1 -23200.393,E2 -23200.393} C_VEL
LIN {X 0,Y 353.179,Z 685.287,A -85,B 0,C 180,E1 -23200.61,E2 -23200.61} C_VEL
LIN {X 0,Y 347.296,Z 739.6,A -85,B 0,C 180,E1 -23202.424,E2 -23202.424} C_VEL
LIN {X 0,Y 345.739,Z 750.365,A -85,B 0,C 180,E1 -23202.925,E2 -23202.925} C_VEL
LIN {X 0,Y 343.829,Z 761.029,A -85,B 0,C 180,E1 -23203.574,E2 -23203.574} C_VEL
LIN {X 0,Y 341.289,Z 773.115,A -85,B 0,C 180,E1 -23204.525,E2 -23204.525} C_VEL
LIN {X 0,Y 338.203,Z 785.384,A -85,B 0,C 180,E1 -23205.762,E2 -23205.762} C_VEL
LIN {X 0,Y 335.301,Z 795.304,A -85,B 0,C 180,E1 -23207.022,E2 -23207.022} C_VEL
LIN {X 0,Y 332.922,Z 802.768,A -85,B 0,C 180,E1 -23208.162,E2 -23208.162} C_VEL
LIN {X 0,Y 330.029,Z 810.67,A -85,B 0,C 180,E1 -23209.607,E2 -23209.607} C_VEL
LIN {X 0,Y 327.358,Z 817.302,A -85,B 0,C 180,E1 -23211.075,E2 -23211.075} C_VEL
LIN {X 0,Y 324.936,Z 822.923,A -85,B 0,C 180,E1 -23212.568,E2 -23212.568} C_VEL
LIN {X 0,Y 322.311,Z 828.392,A -85,B 0,C 180,E1 -23214.387,E2 -23214.387} C_VEL
LIN {X 0,Y 320.039,Z 832.672,A -85,B 0,C 180,E1 -23216.235,E2 -23216.235} C_VEL
LIN {X 0,Y 318.743,Z 834.961,A -85,B 0,C 180,E1 -23217.481,E2 -23217.481} C_VEL
LIN {X 0,Y 316.699,Z 838.071,A -85,B 0,C 180,E1 -23220,E2 -23220} C_VEL
LIN {X 0,Y 315.439,Z 839.407,A -85,B 0,C 180,E1 -23222.223,E2 -23222.223} C_VEL
LIN {X 0,Y 314.74,Z 839.672,A -85,B 0,C 180,E1 -23223.828,E2 -23223.828} C_VEL
LIN {X 0,Y 313.952,Z 838.54,A -85,B 0,C 180,E1 -23226.404,E2 -23226.404} C_VEL
LIN {X 0,Y 313.759,Z 837.451,A -85,B 0,C 180,E1 -23227.697,E2 -23227.697} C_VEL
LIN {X 0,Y 313.698,Z 834.88,A -85,B 0,C 180,E1 -23229.64,E2 -23229.64} C_VEL
LIN {X 0,Y 313.714,Z 831.223,A -85,B 0,C 180,E1 -23231.592,E2 -23231.592} C_VEL
LIN {X 0,Y 313.888,Z 825.381,A -85,B 0,C 180,E1 -23233.879,E2 -23233.879} C_VEL
LIN {X 0,Y 314.273,Z 819.03,A -85,B 0,C 180,E1 -23235.803,E2 -23235.803} C_VEL
LIN {X 0,Y 314.597,Z 812.185,A -85,B 0,C 180,E1 -23237.492,E2 -23237.492} C_VEL
LIN {X 0,Y 314.92,Z 805.873,A -85,B 0,C 180,E1 -23238.814,E2 -23238.814} C_VEL
LIN {X 0,Y 315.513,Z 796.355,A -85,B 0,C 180,E1 -23240.465,E2 -23240.465} C_VEL
LIN {X 0,Y 316.042,Z 787.623,A -85,B 0,C 180,E1 -23241.729,E2 -23241.729} C_VEL
LIN {X 0,Y 316.548,Z 779.04,A -85,B 0,C 180,E1 -23242.782,E2 -23242.782} C_VEL
LIN {X 0,Y 317.199,Z 769.47,A -85,B 0,C 180,E1 -23243.765,E2 -23243.765} C_VEL
LIN {X 0,Y 317.72,Z 758.546,A -85,B 0,C 180,E1 -23244.676,E2 -23244.676} C_VEL
LIN {X 0,Y 318.156,Z 747.506,A -85,B 0,C 180,E1 -23245.4,E2 -23245.4} C_VEL
LIN {X 0,Y 318.599,Z 736.504,A -85,B 0,C 180,E1 -23245.944,E2 -23245.944} C_VEL
LIN {X 0,Y 319.882,Z 695.432,A -85,B 0,C 180,E1 -23247.332,E2 -23247.332} C_VEL
LIN {X 0,Y 320.872,Z 661.483,A -85,B 0,C 180,E1 -23248.454,E2 -23248.454} C_VEL
LIN {X 0,Y 318.058,Z 634.347,A -85,B 0,C 180,E1 -23249.43,E2 -23249.43} C_VEL
LIN {X 0,Y 317.655,Z 628.474,A -85,B 0,C 180,E1 -23249.661,E2 -23249.661} C_VEL
LIN {X 0,Y 318.054,Z 624.804,A -85,B 0,C 180,E1 -23250.807,E2 -23250.807} C_VEL
LIN {X 0,Y 316.874,Z 617.943,A -85,B 0,C 180,E1 -23253.062,E2 -23253.062} C_VEL
LIN {X 0,Y 316.656,Z 617.968,A -85,B 0,C 180,E1 -23257.219,E2 -23257.219} C_VEL
LIN {X 0,Y 316.625,Z 617.974,A -85,B 0,C 180,E1 -23261.222,E2 -23261.222} C_VEL
LIN {X 0,Y 316.655,Z 617.969,A -85,B 0,C 180,E1 -23265.059,E2 -23265.059} C_VEL
LIN {X 0,Y 316.624,Z 617.974,A -85,B 0,C 180,E1 -23268.776,E2 -23268.776} C_VEL
LIN {X 0,Y 316.652,Z 617.971,A -85,B 0,C 180,E1 -23272.78,E2 -23272.78} C_VEL
LIN {X 0,Y 316.63,Z 617.974,A -85,B 0,C 180,E1 -23276.423,E2 -23276.423} C_VEL
LIN {X 0,Y 316.644,Z 617.974,A -85,B 0,C 180,E1 -23279.621,E2 -23279.621} C_VEL
LIN {X 0,Y 316.696,Z 617.968,A -85,B 0,C 180,E1 -23283.746,E2 -23283.746} C_VEL
LIN {X 0,Y 316.705,Z 617.968,A -85,B 0,C 180,E1 -23287.915,E2 -23287.915} C_VEL
LIN {X 0,Y 316.768,Z 617.962,A -85,B 0,C 180,E1 -23291.966,E2 -23291.966} C_VEL
LIN {X 0,Y 316.893,Z 617.941,A -85,B 0,C 180,E1 -23296.542,E2 -23296.542} C_VEL
LIN {X 0,Y 316.939,Z 617.935,A -85,B 0,C 180,E1 -23301.1,E2 -23301.1} C_VEL
LIN {X 0,Y 317.118,Z 617.915,A -85,B 0,C 180,E1 -23303.688,E2 -23303.688} C_VEL
LIN {X 0,Y 317.109,Z 617.914,A -85,B 0,C 180,E1 -23307.468,E2 -23307.468} C_VEL
LIN {X 0,Y 317.139,Z 617.911,A -85,B 0,C 180,E1 -23311.265,E2 -23311.265} C_VEL
LIN {X 0,Y 317.089,Z 617.914,A -85,B 0,C 180,E1 -23315.069,E2 -23315.069} C_VEL
LIN {X 0,Y 316.992,Z 617.93,A -85,B 0,C 180,E1 -23317.618,E2 -23317.618} C_VEL
LIN {X 0,Y 316.837,Z 617.949,A -85,B 0,C 180,E1 -23321.476,E2 -23321.476} C_VEL
LIN {X 0,Y 316.832,Z 617.951,A -85,B 0,C 180,E1 -23324.074,E2 -23324.074} C_VEL
LIN {X 0,Y 316.773,Z 617.961,A -85,B 0,C 180,E1 -23328.048,E2 -23328.048} C_VEL
LIN {X 0,Y 316.704,Z 617.968,A -85,B 0,C 180,E1 -23332.085,E2 -23332.085} C_VEL
LIN {X 0,Y 316.694,Z 617.968,A -85,B 0,C 180,E1 -23336.253,E2 -23336.253} C_VEL
LIN {X 0,Y 316.649,Z 617.973,A -85,B 0,C 180,E1 -23340.38,E2 -23340.38} C_VEL
LIN {X 0,Y 316.684,Z 617.967,A -85,B 0,C 180,E1 -23343.569,E2 -23343.569} C_VEL
LIN {X 0,Y 316.723,Z 617.962,A -85,B 0,C 180,E1 -23347.237,E2 -23347.237} C_VEL
LIN {X 0,Y 316.681,Z 617.967,A -85,B 0,C 180,E1 -23351.235,E2 -23351.235} C_VEL
LIN {X 0,Y 316.653,Z 617.969,A -85,B 0,C 180,E1 -23355.06,E2 -23355.06} C_VEL
LIN {X 0,Y 316.681,Z 617.968,A -85,B 0,C 180,E1 -23358.766,E2 -23358.766} C_VEL
LIN {X 0,Y 316.69,Z 617.964,A -85,B 0,C 180,E1 -23362.772,E2 -23362.772} C_VEL
LIN {X 0,Y 316.633,Z 617.975,A -85,B 0,C 180,E1 -23366.425,E2 -23366.425} C_VEL
LIN {X 0,Y 316.645,Z 617.974,A -85,B 0,C 180,E1 -23369.622,E2 -23369.622} C_VEL
LIN {X 0,Y 316.696,Z 617.966,A -85,B 0,C 180,E1 -23373.747,E2 -23373.747} C_VEL
LIN {X 0,Y 316.706,Z 617.969,A -85,B 0,C 180,E1 -23377.916,E2 -23377.916} C_VEL
LIN {X 0,Y 316.751,Z 617.962,A -85,B 0,C 180,E1 -23381.966,E2 -23381.966} C_VEL
LIN {X 0,Y 316.844,Z 617.948,A -85,B 0,C 180,E1 -23386.582,E2 -23386.582} C_VEL
LIN {X 0,Y 316.945,Z 617.933,A -85,B 0,C 180,E1 -23391.101,E2 -23391.101} C_VEL
LIN {X 0,Y 317.158,Z 617.908,A -85,B 0,C 180,E1 -23393.661,E2 -23393.661} C_VEL
LIN {X 0,Y 317.113,Z 617.915,A -85,B 0,C 180,E1 -23397.468,E2 -23397.468} C_VEL
LIN {X 0,Y 317.14,Z 617.909,A -85,B 0,C 180,E1 -23401.266,E2 -23401.266} C_VEL
LIN {X 0,Y 317.089,Z 617.916,A -85,B 0,C 180,E1 -23405.07,E2 -23405.07} C_VEL
LIN {X 0,Y 316.996,Z 617.93,A -85,B 0,C 180,E1 -23407.619,E2 -23407.619} C_VEL
LIN {X 0,Y 316.833,Z 617.948,A -85,B 0,C 180,E1 -23411.477,E2 -23411.477} C_VEL
LIN {X 0,Y 316.781,Z 617.959,A -85,B 0,C 180,E1 -23414.077,E2 -23414.077} C_VEL
LIN {X 0,Y 316.717,Z 617.968,A -85,B 0,C 180,E1 -23418.037,E2 -23418.037} C_VEL
LIN {X 0,Y 316.677,Z 617.971,A -85,B 0,C 180,E1 -23422.087,E2 -23422.087} C_VEL
LIN {X 0,Y 316.698,Z 617.968,A -85,B 0,C 180,E1 -23426.254,E2 -23426.254} C_VEL
LIN {X 0,Y 316.645,Z 617.971,A -85,B 0,C 180,E1 -23429.121,E2 -23429.121} C_VEL
LIN {X 0,Y 316.639,Z 617.971,A -85,B 0,C 180,E1 -23432.796,E2 -23432.796} C_VEL
LIN {X 0,Y 316.617,Z 617.972,A -85,B 0,C 180,E1 -23434.427,E2 -23434.427} C_VEL
LIN {X 0,Y 315.983,Z 618.056,A -85,B 0,C 180,E1 -23435.488,E2 -23435.488} C_VEL
LIN {X 0,Y 313.142,Z 618.413,A -85,B 0,C 180,E1 -23437.215,E2 -23437.215} C_VEL
LIN {X 0,Y 310.706,Z 618.717,A -85,B 0,C 180,E1 -23438.616,E2 -23438.616} C_VEL
LIN {X 0,Y 309.647,Z 618.846,A -85,B 0,C 180,E1 -23439.7,E2 -23439.7} C_VEL
LIN {X 0,Y 309.555,Z 618.854,A -85,B 0,C 180,E1 -23440.068,E2 -23440.068} C_VEL
LIN {X 0,Y 309.577,Z 618.853,A -85,B 0,C 180,E1 -23443.612,E2 -23443.612} C_VEL
LIN {X 0,Y 309.57,Z 618.853,A -85,B 0,C 180,E1 -23447.251,E2 -23447.251} C_VEL
LIN {X 0,Y 309.566,Z 618.851,A -85,B 0,C 180,E1 -23450.688,E2 -23450.688} C_VEL
LIN {X 0,Y 309.585,Z 618.852,A -85,B 0,C 180,E1 -23454.539,E2 -23454.539} C_VEL
LIN {X 0,Y 309.608,Z 618.848,A -85,B 0,C 180,E1 -23457.114,E2 -23457.114} C_VEL
LIN {X 0,Y 309.643,Z 618.843,A -85,B 0,C 180,E1 -23461.638,E2 -23461.638} C_VEL
LIN {X 0,Y 309.771,Z 618.918,A -85,B 0,C 180,E1 -23462.977,E2 -23462.977} C_VEL
LIN {X 0,Y 311.588,Z 629.051,A -85,B 0,C 180,E1 -23466.132,E2 -23466.132} C_VEL
LIN {X 0,Y 311.806,Z 631.044,A -85,B 0,C 180,E1 -23466.739,E2 -23466.739} C_VEL
LIN {X 0,Y 310.204,Z 642.864,A -85,B 0,C 180,E1 -23470.202,E2 -23470.202} C_VEL
LIN {X 0,Y 311.523,Z 665.789,A -85,B 0,C 180,E1 -23471.027,E2 -23471.027} C_VEL
LIN {X 0,Y 313.418,Z 687.452,A -85,B 0,C 180,E1 -23471.809,E2 -23471.809} C_VEL
LIN {X 0,Y 311.639,Z 748.542,A -85,B 0,C 180,E1 -23473.935,E2 -23473.935} C_VEL
LIN {X 0,Y 311.151,Z 759.433,A -85,B 0,C 180,E1 -23474.453,E2 -23474.453} C_VEL
LIN {X 0,Y 310.795,Z 769.142,A -85,B 0,C 180,E1 -23475.063,E2 -23475.063} C_VEL
LIN {X 0,Y 310.326,Z 779.469,A -85,B 0,C 180,E1 -23475.881,E2 -23475.881} C_VEL
LIN {X 0,Y 309.807,Z 788.742,A -85,B 0,C 180,E1 -23476.78,E2 -23476.78} C_VEL
LIN {X 0,Y 309.087,Z 798.299,A -85,B 0,C 180,E1 -23477.9,E2 -23477.9} C_VEL
LIN {X 0,Y 308.6,Z 806.536,A -85,B 0,C 180,E1 -23479.042,E2 -23479.042} C_VEL
LIN {X 0,Y 308.082,Z 815.394,A -85,B 0,C 180,E1 -23480.513,E2 -23480.513} C_VEL
LIN {X 0,Y 307.684,Z 822.113,A -85,B 0,C 180,E1 -23481.82,E2 -23481.82} C_VEL
LIN {X 0,Y 307.451,Z 829.185,A -85,B 0,C 180,E1 -23483.459,E2 -23483.459} C_VEL
LIN {X 0,Y 307.282,Z 835.071,A -85,B 0,C 180,E1 -23485.097,E2 -23485.097} C_VEL
LIN {X 0,Y 307.161,Z 839.934,A -85,B 0,C 180,E1 -23486.732,E2 -23486.732} C_VEL
LIN {X 0,Y 307.1,Z 844.531,A -85,B 0,C 180,E1 -23488.693,E2 -23488.693} C_VEL
LIN {X 0,Y 307.009,Z 846.845,A -85,B 0,C 180,E1 -23490,E2 -23490} C_VEL
LIN {X 0,Y 306.971,Z 848.749,A -85,B 0,C 180,E1 -23491.308,E2 -23491.308} C_VEL
LIN {X 0,Y 306.873,Z 850.306,A -85,B 0,C 180,E1 -23492.617,E2 -23492.617} C_VEL
LIN {X 0,Y 306.95,Z 851.908,A -85,B 0,C 180,E1 -23495.237,E2 -23495.237} C_VEL
LIN {X 0,Y 307.183,Z 852.157,A -85,B 0,C 180,E1 -23496.547,E2 -23496.547} C_VEL
LIN {X 0,Y 308.043,Z 851.404,A -85,B 0,C 180,E1 -23499.159,E2 -23499.159} C_VEL
LIN {X 0,Y 309.695,Z 848.943,A -85,B 0,C 180,E1 -23501.745,E2 -23501.745} C_VEL
LIN {X 0,Y 311.375,Z 846.058,A -85,B 0,C 180,E1 -23503.663,E2 -23503.663} C_VEL
LIN {X 0,Y 313.437,Z 842.148,A -85,B 0,C 180,E1 -23505.555,E2 -23505.555} C_VEL
LIN {X 0,Y 315.739,Z 837.604,A -85,B 0,C 180,E1 -23507.255,E2 -23507.255} C_VEL
LIN {X 0,Y 318.16,Z 832.211,A -85,B 0,C 180,E1 -23508.916,E2 -23508.916} C_VEL
LIN {X 0,Y 321.495,Z 824.65,A -85,B 0,C 180,E1 -23510.735,E2 -23510.735} C_VEL
LIN {X 0,Y 324.364,Z 817.243,A -85,B 0,C 180,E1 -23512.204,E2 -23512.204} C_VEL
LIN {X 0,Y 327.544,Z 808.355,A -85,B 0,C 180,E1 -23513.639,E2 -23513.639} C_VEL
LIN {X 0,Y 330.697,Z 798.82,A -85,B 0,C 180,E1 -23514.896,E2 -23514.896} C_VEL
LIN {X 0,Y 333.327,Z 790.112,A -85,B 0,C 180,E1 -23515.851,E2 -23515.851} C_VEL
LIN {X 0,Y 335.732,Z 781.329,A -85,B 0,C 180,E1 -23516.652,E2 -23516.652} C_VEL
LIN {X 0,Y 338.26,Z 770.699,A -85,B 0,C 180,E1 -23517.435,E2 -23517.435} C_VEL
LIN {X 0,Y 340.406,Z 759.71,A -85,B 0,C 180,E1 -23518.08,E2 -23518.08} C_VEL
LIN {X 0,Y 342.109,Z 749.107,A -85,B 0,C 180,E1 -23518.552,E2 -23518.552} C_VEL
LIN {X 0,Y 347.264,Z 702.353,A -85,B 0,C 180,E1 -23520.175,E2 -23520.175} C_VEL
LIN {X 0,Y 346.081,Z 690.809,A -85,B 0,C 180,E1 -23521.111,E2 -23521.111} C_VEL
LIN {X 0,Y 345.619,Z 688.577,A -85,B 0,C 180,E1 -23521.35,E2 -23521.35} C_VEL
LIN {X 0,Y 341.829,Z 679.587,A -85,B 0,C 180,E1 -23522.846,E2 -23522.846} C_VEL
LIN {X 0,Y 338.316,Z 672.48,A -85,B 0,C 180,E1 -23524.303,E2 -23524.303} C_VEL
LIN {X 0,Y 335.527,Z 667.229,A -85,B 0,C 180,E1 -23525.583,E2 -23525.583} C_VEL
LIN {X 0,Y 332.989,Z 662.725,A -85,B 0,C 180,E1 -23526.813,E2 -23526.813} C_VEL
LIN {X 0,Y 330.155,Z 657.716,A -85,B 0,C 180,E1 -23528.407,E2 -23528.407} C_VEL
LIN {X 0,Y 326.625,Z 652.543,A -85,B 0,C 180,E1 -23530.652,E2 -23530.652} C_VEL
LIN {X 0,Y 325.576,Z 650.826,A -85,B 0,C 180,E1 -23531.458,E2 -23531.458} C_VEL
LIN {X 0,Y 321.585,Z 644.86,A -85,B 0,C 180,E1 -23535.705,E2 -23535.705} C_VEL
LIN {X 0,Y 320.836,Z 643.531,A -85,B 0,C 180,E1 -23537.184,E2 -23537.184} C_VEL
LIN {X 0,Y 320.182,Z 642.581,A -85,B 0,C 180,E1 -23539.968,E2 -23539.968} C_VEL
LIN {X 0,Y 320.697,Z 642.631,A -85,B 0,C 180,E1 -23542.692,E2 -23542.692} C_VEL
LIN {X 0,Y 321.95,Z 644.567,A -85,B 0,C 180,E1 -23545.173,E2 -23545.173} C_VEL
LIN {X 0,Y 325.36,Z 648.124,A -85,B 0,C 180,E1 -23548.564,E2 -23548.564} C_VEL
LIN {X 0,Y 328.436,Z 652.439,A -85,B 0,C 180,E1 -23550.807,E2 -23550.807} C_VEL
LIN {X 0,Y 329.437,Z 653.706,A -85,B 0,C 180,E1 -23551.398,E2 -23551.398} C_VEL
LIN {X 0,Y 333.005,Z 659.034,A -85,B 0,C 180,E1 -23553.395,E2 -23553.395} C_VEL
LIN {X 0,Y 336.537,Z 664.482,A -85,B 0,C 180,E1 -23555.052,E2 -23555.052} C_VEL
LIN {X 0,Y 339.322,Z 669.188,A -85,B 0,C 180,E1 -23556.264,E2 -23556.264} C_VEL
LIN {X 0,Y 343.031,Z 675.929,A -85,B 0,C 180,E1 -23557.74,E2 -23557.74} C_VEL
LIN {X 0,Y 347.44,Z 685.257,A -85,B 0,C 180,E1 -23559.373,E2 -23559.373} C_VEL
LIN {X 0,Y 348.556,Z 687.961,A -85,B 0,C 180,E1 -23559.781,E2 -23559.781} C_VEL
LIN {X 0,Y 342.512,Z 740.041,A -85,B 0,C 180,E1 -23561.558,E2 -23561.558} C_VEL
LIN {X 0,Y 340.717,Z 751.825,A -85,B 0,C 180,E1 -23562.116,E2 -23562.116} C_VEL
LIN {X 0,Y 338.536,Z 763.401,A -85,B 0,C 180,E1 -23562.852,E2 -23562.852} C_VEL
LIN {X 0,Y 335.707,Z 775.666,A -85,B 0,C 180,E1 -23563.869,E2 -23563.869} C_VEL
LIN {X 0,Y 332.635,Z 786.735,A -85,B 0,C 180,E1 -23565.051,E2 -23565.051} C_VEL
LIN {X 0,Y 329.893,Z 795.426,A -85,B 0,C 180,E1 -23566.18,E2 -23566.18} C_VEL
LIN {X 0,Y 327.393,Z 802.902,A -85,B 0,C 180,E1 -23567.332,E2 -23567.332} C_VEL
LIN {X 0,Y 324.367,Z 810.831,A -85,B 0,C 180,E1 -23568.793,E2 -23568.793} C_VEL
LIN {X 0,Y 321.529,Z 817.498,A -85,B 0,C 180,E1 -23570.28,E2 -23570.28} C_VEL
LIN {X 0,Y 318.766,Z 823.414,A -85,B 0,C 180,E1 -23571.897,E2 -23571.897} C_VEL
LIN {X 0,Y 316.14,Z 828.515,A -85,B 0,C 180,E1 -23573.639,E2 -23573.639} C_VEL
LIN {X 0,Y 313.706,Z 832.823,A -85,B 0,C 180,E1 -23575.517,E2 -23575.517} C_VEL
LIN {X 0,Y 311.643,Z 836.049,A -85,B 0,C 180,E1 -23577.423,E2 -23577.423} C_VEL
LIN {X 0,Y 310.515,Z 837.635,A -85,B 0,C 180,E1 -23578.707,E2 -23578.707} C_VEL
LIN {X 0,Y 308.782,Z 839.537,A -85,B 0,C 180,E1 -23581.299,E2 -23581.299} C_VEL
LIN {X 0,Y 307.594,Z 839.693,A -85,B 0,C 180,E1 -23583.917,E2 -23583.917} C_VEL
LIN {X 0,Y 307.151,Z 839.265,A -85,B 0,C 180,E1 -23585.233,E2 -23585.233} C_VEL
LIN {X 0,Y 306.656,Z 836.907,A -85,B 0,C 180,E1 -23587.877,E2 -23587.877} C_VEL
LIN {X 0,Y 306.631,Z 834.035,A -85,B 0,C 180,E1 -23589.864,E2 -23589.864} C_VEL
LIN {X 0,Y 306.637,Z 830.046,A -85,B 0,C 180,E1 -23591.863,E2 -23591.863} C_VEL
LIN {X 0,Y 306.826,Z 824.824,A -85,B 0,C 180,E1 -23593.868,E2 -23593.868} C_VEL
LIN {X 0,Y 307.174,Z 819.42,A -85,B 0,C 180,E1 -23595.541,E2 -23595.541} C_VEL
LIN {X 0,Y 307.457,Z 812.796,A -85,B 0,C 180,E1 -23597.227,E2 -23597.227} C_VEL
LIN {X 0,Y 307.896,Z 804.769,A -85,B 0,C 180,E1 -23598.915,E2 -23598.915} C_VEL
LIN {X 0,Y 308.375,Z 797.153,A -85,B 0,C 180,E1 -23600.266,E2 -23600.266} C_VEL
LIN {X 0,Y 308.916,Z 788.076,A -85,B 0,C 180,E1 -23601.619,E2 -23601.619} C_VEL
LIN {X 0,Y 309.488,Z 778.572,A -85,B 0,C 180,E1 -23602.803,E2 -23602.803} C_VEL
LIN {X 0,Y 310.141,Z 768.865,A -85,B 0,C 180,E1 -23603.809,E2 -23603.809} C_VEL
LIN {X 0,Y 310.601,Z 758.895,A -85,B 0,C 180,E1 -23604.657,E2 -23604.657} C_VEL
LIN {X 0,Y 311.044,Z 748.356,A -85,B 0,C 180,E1 -23605.373,E2 -23605.373} C_VEL
LIN {X 0,Y 311.482,Z 737.013,A -85,B 0,C 180,E1 -23605.955,E2 -23605.955} C_VEL
LIN {X 0,Y 312.643,Z 703.097,A -85,B 0,C 180,E1 -23607.16,E2 -23607.16} C_VEL
LIN {X 0,Y 313.727,Z 661.391,A -85,B 0,C 180,E1 -23608.592,E2 -23608.592} C_VEL
LIN {X 0,Y 310.78,Z 632.081,A -85,B 0,C 180,E1 -23609.664,E2 -23609.664} C_VEL
LIN {X 0,Y 310.624,Z 628.561,A -85,B 0,C 180,E1 -23609.834,E2 -23609.834} C_VEL
LIN {X 0,Y 310.861,Z 624.612,A -85,B 0,C 180,E1 -23611.103,E2 -23611.103} C_VEL
LIN {X 0,Y 309.819,Z 618.822,A -85,B 0,C 180,E1 -23613.048,E2 -23613.048} C_VEL
LIN {X 0,Y 309.607,Z 618.848,A -85,B 0,C 180,E1 -23617.649,E2 -23617.649} C_VEL
LIN {X 0,Y 309.59,Z 618.854,A -85,B 0,C 180,E1 -23621.701,E2 -23621.701} C_VEL
LIN {X 0,Y 309.606,Z 618.848,A -85,B 0,C 180,E1 -23625.465,E2 -23625.465} C_VEL
LIN {X 0,Y 309.588,Z 618.85,A -85,B 0,C 180,E1 -23628.994,E2 -23628.994} C_VEL
LIN {X 0,Y 309.605,Z 618.851,A -85,B 0,C 180,E1 -23632.356,E2 -23632.356} C_VEL
LIN {X 0,Y 309.578,Z 618.852,A -85,B 0,C 180,E1 -23635.553,E2 -23635.553} C_VEL
LIN {X 0,Y 309.602,Z 618.849,A -85,B 0,C 180,E1 -23639.283,E2 -23639.283} C_VEL
LIN {X 0,Y 309.636,Z 618.844,A -85,B 0,C 180,E1 -23643.1,E2 -23643.1} C_VEL
LIN {X 0,Y 309.631,Z 618.848,A -85,B 0,C 180,E1 -23645.971,E2 -23645.971} C_VEL
LIN {X 0,Y 309.68,Z 618.839,A -85,B 0,C 180,E1 -23648.783,E2 -23648.783} C_VEL
LIN {X 0,Y 309.712,Z 618.835,A -85,B 0,C 180,E1 -23652.902,E2 -23652.902} C_VEL
LIN {X 0,Y 309.842,Z 618.818,A -85,B 0,C 180,E1 -23656.934,E2 -23656.934} C_VEL
LIN {X 0,Y 309.899,Z 618.812,A -85,B 0,C 180,E1 -23660.896,E2 -23660.896} C_VEL
LIN {X 0,Y 310.078,Z 618.792,A -85,B 0,C 180,E1 -23663.677,E2 -23663.677} C_VEL
LIN {X 0,Y 310.066,Z 618.791,A -85,B 0,C 180,E1 -23667.41,E2 -23667.41} C_VEL
LIN {X 0,Y 310.117,Z 618.785,A -85,B 0,C 180,E1 -23671.294,E2 -23671.294} C_VEL
LIN {X 0,Y 310.04,Z 618.792,A -85,B 0,C 180,E1 -23675.185,E2 -23675.185} C_VEL
LIN {X 0,Y 309.958,Z 618.807,A -85,B 0,C 180,E1 -23677.792,E2 -23677.792} C_VEL
LIN {X 0,Y 309.794,Z 618.828,A -85,B 0,C 180,E1 -23681.741,E2 -23681.741} C_VEL
LIN {X 0,Y 309.765,Z 618.828,A -85,B 0,C 180,E1 -23684.402,E2 -23684.402} C_VEL
LIN {X 0,Y 309.713,Z 618.837,A -85,B 0,C 180,E1 -23688.459,E2 -23688.459} C_VEL
LIN {X 0,Y 309.683,Z 618.843,A -85,B 0,C 180,E1 -23691.978,E2 -23691.978} C_VEL
LIN {X 0,Y 309.647,Z 618.842,A -85,B 0,C 180,E1 -23695.454,E2 -23695.454} C_VEL
LIN {X 0,Y 309.605,Z 618.851,A -85,B 0,C 180,E1 -23698.366,E2 -23698.366} C_VEL
LIN {X 0,Y 309.604,Z 618.849,A -85,B 0,C 180,E1 -23701.355,E2 -23701.355} C_VEL
LIN {X 0,Y 309.625,Z 618.846,A -85,B 0,C 180,E1 -23704.441,E2 -23704.441} C_VEL
LIN {X 0,Y 309.675,Z 618.842,A -85,B 0,C 180,E1 -23707.661,E2 -23707.661} C_VEL
LIN {X 0,Y 309.638,Z 618.847,A -85,B 0,C 180,E1 -23711.712,E2 -23711.712} C_VEL
LIN {X 0,Y 309.605,Z 618.848,A -85,B 0,C 180,E1 -23715.467,E2 -23715.467} C_VEL
LIN {X 0,Y 309.639,Z 618.845,A -85,B 0,C 180,E1 -23719.004,E2 -23719.004} C_VEL
LIN {X 0,Y 309.638,Z 618.844,A -85,B 0,C 180,E1 -23722.355,E2 -23722.355} C_VEL
LIN {X 0,Y 309.59,Z 618.851,A -85,B 0,C 180,E1 -23725.555,E2 -23725.555} C_VEL
LIN {X 0,Y 309.602,Z 618.85,A -85,B 0,C 180,E1 -23729.284,E2 -23729.284} C_VEL
LIN {X 0,Y 309.637,Z 618.842,A -85,B 0,C 180,E1 -23733.101,E2 -23733.101} C_VEL
LIN {X 0,Y 309.633,Z 618.849,A -85,B 0,C 180,E1 -23735.972,E2 -23735.972} C_VEL
LIN {X 0,Y 309.682,Z 618.839,A -85,B 0,C 180,E1 -23738.784,E2 -23738.784} C_VEL
LIN {X 0,Y 309.69,Z 618.835,A -85,B 0,C 180,E1 -23742.901,E2 -23742.901} C_VEL
LIN {X 0,Y 309.813,Z 618.823,A -85,B 0,C 180,E1 -23746.934,E2 -23746.934} C_VEL
LIN {X 0,Y 309.904,Z 618.81,A -85,B 0,C 180,E1 -23750.897,E2 -23750.897} C_VEL
LIN {X 0,Y 310.128,Z 618.783,A -85,B 0,C 180,E1 -23753.598,E2 -23753.598} C_VEL
LIN {X 0,Y 310.071,Z 618.792,A -85,B 0,C 180,E1 -23757.411,E2 -23757.411} C_VEL
LIN {X 0,Y 310.118,Z 618.784,A -85,B 0,C 180,E1 -23761.295,E2 -23761.295} C_VEL
LIN {X 0,Y 310.041,Z 618.794,A -85,B 0,C 180,E1 -23765.185,E2 -23765.185} C_VEL
LIN {X 0,Y 309.961,Z 618.808,A -85,B 0,C 180,E1 -23767.793,E2 -23767.793} C_VEL
LIN {X 0,Y 309.787,Z 618.827,A -85,B 0,C 180,E1 -23771.742,E2 -23771.742} C_VEL
LIN {X 0,Y 309.707,Z 618.838,A -85,B 0,C 180,E1 -23774.406,E2 -23774.406} C_VEL
LIN {X 0,Y 309.658,Z 618.843,A -85,B 0,C 180,E1 -23778.463,E2 -23778.463} C_VEL
LIN {X 0,Y 309.617,Z 618.846,A -85,B 0,C 180,E1 -23782.619,E2 -23782.619} C_VEL
LIN {X 0,Y 309.651,Z 618.844,A -85,B 0,C 180,E1 -23785.454,E2 -23785.454} C_VEL
LIN {X 0,Y 309.605,Z 618.85,A -85,B 0,C 180,E1 -23788.366,E2 -23788.366} C_VEL
LIN {X 0,Y 309.553,Z 618.853,A -85,B 0,C 180,E1 -23791.362,E2 -23791.362} C_VEL
LIN {X 0,Y 309.576,Z 618.854,A -85,B 0,C 180,E1 -23794.448,E2 -23794.448} C_VEL
LIN {X 0,Y 309.589,Z 618.853,A -85,B 0,C 180,E1 -23797.653,E2 -23797.653} C_VEL
LIN {X 0,Y 309.555,Z 618.854,A -85,B 0,C 180,E1 -23800.068,E2 -23800.068} C_VEL
LIN {X 0,Y 308.86,Z 618.939,A -85,B 0,C 180,E1 -23801.153,E2 -23801.153} C_VEL
LIN {X 0,Y 305.966,Z 619.301,A -85,B 0,C 180,E1 -23802.92,E2 -23802.92} C_VEL
LIN {X 0,Y 303.557,Z 619.604,A -85,B 0,C 180,E1 -23804.353,E2 -23804.353} C_VEL
LIN {X 0,Y 302.571,Z 619.727,A -85,B 0,C 180,E1 -23805.464,E2 -23805.464} C_VEL
LIN {X 0,Y 302.516,Z 619.736,A -85,B 0,C 180,E1 -23805.84,E2 -23805.84} C_VEL
LIN {X 0,Y 302.53,Z 619.733,A -85,B 0,C 180,E1 -23809.822,E2 -23809.822} C_VEL
LIN {X 0,Y 302.531,Z 619.729,A -85,B 0,C 180,E1 -23812.989,E2 -23812.989} C_VEL
LIN {X 0,Y 302.532,Z 619.731,A -85,B 0,C 180,E1 -23816.46,E2 -23816.46} C_VEL
LIN {X 0,Y 302.55,Z 619.727,A -85,B 0,C 180,E1 -23819.381,E2 -23819.381} C_VEL
LIN {X 0,Y 302.733,Z 619.895,A -85,B 0,C 180,E1 -23822.995,E2 -23822.995} C_VEL
LIN {X 0,Y 304.57,Z 630.18,A -85,B 0,C 180,E1 -23826.269,E2 -23826.269} C_VEL
LIN {X 0,Y 304.426,Z 633.635,A -85,B 0,C 180,E1 -23827.332,E2 -23827.332} C_VEL
LIN {X 0,Y 303.139,Z 642.527,A -85,B 0,C 180,E1 -23830.04,E2 -23830.04} C_VEL
LIN {X 0,Y 304.257,Z 664.068,A -85,B 0,C 180,E1 -23830.844,E2 -23830.844} C_VEL
LIN {X 0,Y 306.342,Z 687.389,A -85,B 0,C 180,E1 -23831.719,E2 -23831.719} C_VEL
LIN {X 0,Y 304.538,Z 749.059,A -85,B 0,C 180,E1 -23833.936,E2 -23833.936} C_VEL
LIN {X 0,Y 304.059,Z 759.743,A -85,B 0,C 180,E1 -23834.467,E2 -23834.467} C_VEL
LIN {X 0,Y 303.643,Z 769.854,A -85,B 0,C 180,E1 -23835.13,E2 -23835.13} C_VEL
LIN {X 0,Y 303.259,Z 778.982,A -85,B 0,C 180,E1 -23835.872,E2 -23835.872} C_VEL
LIN {X 0,Y 302.625,Z 789.766,A -85,B 0,C 180,E1 -23836.958,E2 -23836.958} C_VEL
LIN {X 0,Y 301.937,Z 799.229,A -85,B 0,C 180,E1 -23838.119,E2 -23838.119} C_VEL
LIN {X 0,Y 301.434,Z 807.283,A -85,B 0,C 180,E1 -23839.287,E2 -23839.287} C_VEL
LIN {X 0,Y 300.99,Z 815.136,A -85,B 0,C 180,E1 -23840.625,E2 -23840.625} C_VEL
LIN {X 0,Y 300.561,Z 823.334,A -85,B 0,C 180,E1 -23842.299,E2 -23842.299} C_VEL
LIN {X 0,Y 300.366,Z 828.955,A -85,B 0,C 180,E1 -23843.641,E2 -23843.641} C_VEL
LIN {X 0,Y 300.221,Z 834.817,A -85,B 0,C 180,E1 -23845.316,E2 -23845.316} C_VEL
LIN {X 0,Y 300.107,Z 840.451,A -85,B 0,C 180,E1 -23847.325,E2 -23847.325} C_VEL
LIN {X 0,Y 300.03,Z 844.835,A -85,B 0,C 180,E1 -23849.331,E2 -23849.331} C_VEL
LIN {X 0,Y 299.909,Z 848.092,A -85,B 0,C 180,E1 -23851.339,E2 -23851.339} C_VEL
LIN {X 0,Y 299.813,Z 849.677,A -85,B 0,C 180,E1 -23852.678,E2 -23852.678} C_VEL
LIN {X 0,Y 299.87,Z 851.628,A -85,B 0,C 180,E1 -23855.361,E2 -23855.361} C_VEL
LIN {X 0,Y 300.467,Z 851.829,A -85,B 0,C 180,E1 -23858.041,E2 -23858.041} C_VEL
LIN {X 0,Y 301.041,Z 851.414,A -85,B 0,C 180,E1 -23859.374,E2 -23859.374} C_VEL
LIN {X 0,Y 302.772,Z 849.282,A -85,B 0,C 180,E1 -23862.018,E2 -23862.018} C_VEL
LIN {X 0,Y 304.516,Z 846.6,A -85,B 0,C 180,E1 -23863.977,E2 -23863.977} C_VEL
LIN {X 0,Y 306.645,Z 842.931,A -85,B 0,C 180,E1 -23865.909,E2 -23865.909} C_VEL
LIN {X 0,Y 309.602,Z 837.487,A -85,B 0,C 180,E1 -23868.039,E2 -23868.039} C_VEL
LIN {X 0,Y 312.722,Z 831.089,A -85,B 0,C 180,E1 -23869.973,E2 -23869.973} C_VEL
LIN {X 0,Y 315.58,Z 824.9,A -85,B 0,C 180,E1 -23871.483,E2 -23871.483} C_VEL
LIN {X 0,Y 318.61,Z 817.587,A -85,B 0,C 180,E1 -23872.969,E2 -23872.969} C_VEL
LIN {X 0,Y 321.965,Z 808.924,A -85,B 0,C 180,E1 -23874.416,E2 -23874.416} C_VEL
LIN {X 0,Y 325.248,Z 799.599,A -85,B 0,C 180,E1 -23875.684,E2 -23875.684} C_VEL
LIN {X 0,Y 327.987,Z 791.045,A -85,B 0,C 180,E1 -23876.646,E2 -23876.646} C_VEL
LIN {X 0,Y 330.911,Z 780.796,A -85,B 0,C 180,E1 -23877.583,E2 -23877.583} C_VEL
LIN {X 0,Y 333.529,Z 770.089,A -85,B 0,C 180,E1 -23878.369,E2 -23878.369} C_VEL
LIN {X 0,Y 335.805,Z 759.108,A -85,B 0,C 180,E1 -23879.01,E2 -23879.01} C_VEL
LIN {X 0,Y 337.443,Z 749.48,A -85,B 0,C 180,E1 -23879.452,E2 -23879.452} C_VEL
LIN {X 0,Y 342.177,Z 709.618,A -85,B 0,C 180,E1 -23880.855,E2 -23880.855} C_VEL
LIN {X 0,Y 342.747,Z 703.484,A -85,B 0,C 180,E1 -23881.099,E2 -23881.099} C_VEL
LIN {X 0,Y 341.753,Z 693.427,A -85,B 0,C 180,E1 -23881.943,E2 -23881.943} C_VEL
LIN {X 0,Y 338.813,Z 685.837,A -85,B 0,C 180,E1 -23883.212,E2 -23883.212} C_VEL
LIN {X 0,Y 335.465,Z 678.62,A -85,B 0,C 180,E1 -23884.678,E2 -23884.678} C_VEL
LIN {X 0,Y 332.046,Z 672.055,A -85,B 0,C 180,E1 -23886.338,E2 -23886.338} C_VEL
LIN {X 0,Y 330.147,Z 668.564,A -85,B 0,C 180,E1 -23887.34,E2 -23887.34} C_VEL
LIN {X 0,Y 327.225,Z 663.35,A -85,B 0,C 180,E1 -23889.087,E2 -23889.087} C_VEL
LIN {X 0,Y 324.105,Z 658.266,A -85,B 0,C 180,E1 -23891.306,E2 -23891.306} C_VEL
LIN {X 0,Y 320.315,Z 652.697,A -85,B 0,C 180,E1 -23895.094,E2 -23895.094} C_VEL
LIN {X 0,Y 319.358,Z 650.604,A -85,B 0,C 180,E1 -23896.938,E2 -23896.938} C_VEL
LIN {X 0,Y 318.64,Z 649.544,A -85,B 0,C 180,E1 -23899.596,E2 -23899.596} C_VEL
LIN {X 0,Y 319.172,Z 649.649,A -85,B 0,C 180,E1 -23902.878,E2 -23902.878} C_VEL
LIN {X 0,Y 320.665,Z 651.962,A -85,B 0,C 180,E1 -23905.631,E2 -23905.631} C_VEL
LIN {X 0,Y 323.43,Z 654.894,A -85,B 0,C 180,E1 -23908.356,E2 -23908.356} C_VEL
LIN {X 0,Y 326.348,Z 659.054,A -85,B 0,C 180,E1 -23910.542,E2 -23910.542} C_VEL
LIN {X 0,Y 327.601,Z 660.956,A -85,B 0,C 180,E1 -23911.349,E2 -23911.349} C_VEL
LIN {X 0,Y 330.413,Z 665.181,A -85,B 0,C 180,E1 -23912.969,E2 -23912.969} C_VEL
LIN {X 0,Y 333.869,Z 670.764,A -85,B 0,C 180,E1 -23914.694,E2 -23914.694} C_VEL
LIN {X 0,Y 337.284,Z 676.78,A -85,B 0,C 180,E1 -23916.244,E2 -23916.244} C_VEL
LIN {X 0,Y 341.146,Z 684.529,A -85,B 0,C 180,E1 -23917.833,E2 -23917.833} C_VEL
LIN {X 0,Y 343.952,Z 691.047,A -85,B 0,C 180,E1 -23918.939,E2 -23918.939} C_VEL
LIN {X 0,Y 337.968,Z 740.218,A -85,B 0,C 180,E1 -23920.634,E2 -23920.634} C_VEL
LIN {X 0,Y 336.215,Z 751.155,A -85,B 0,C 180,E1 -23921.16,E2 -23921.16} C_VEL
LIN {X 0,Y 334.055,Z 761.844,A -85,B 0,C 180,E1 -23921.826,E2 -23921.826} C_VEL
LIN {X 0,Y 330.822,Z 775.676,A -85,B 0,C 180,E1 -23922.955,E2 -23922.955} C_VEL
LIN {X 0,Y 327.807,Z 786.14,A -85,B 0,C 180,E1 -23924.059,E2 -23924.059} C_VEL
LIN {X 0,Y 324.635,Z 795.778,A -85,B 0,C 180,E1 -23925.314,E2 -23925.314} C_VEL
LIN {X 0,Y 321.979,Z 803.179,A -85,B 0,C 180,E1 -23926.475,E2 -23926.475} C_VEL
LIN {X 0,Y 318.771,Z 811.018,A -85,B 0,C 180,E1 -23927.951,E2 -23927.951} C_VEL
LIN {X 0,Y 315.808,Z 817.678,A -85,B 0,C 180,E1 -23929.456,E2 -23929.456} C_VEL
LIN {X 0,Y 313.024,Z 823.305,A -85,B 0,C 180,E1 -23930.988,E2 -23930.988} C_VEL
LIN {X 0,Y 310.071,Z 828.739,A -85,B 0,C 180,E1 -23932.863,E2 -23932.863} C_VEL
LIN {X 0,Y 307.46,Z 833.007,A -85,B 0,C 180,E1 -23934.771,E2 -23934.771} C_VEL
LIN {X 0,Y 305.897,Z 835.283,A -85,B 0,C 180,E1 -23936.061,E2 -23936.061} C_VEL
LIN {X 0,Y 303.423,Z 838.457,A -85,B 0,C 180,E1 -23938.677,E2 -23938.677} C_VEL
LIN {X 0,Y 302.433,Z 839.37,A -85,B 0,C 180,E1 -23940,E2 -23940} C_VEL
LIN {X 0,Y 300.995,Z 840.08,A -85,B 0,C 180,E1 -23942.667,E2 -23942.667} C_VEL
LIN {X 0,Y 300.003,Z 839.017,A -85,B 0,C 180,E1 -23945.358,E2 -23945.358} C_VEL
LIN {X 0,Y 299.689,Z 837.928,A -85,B 0,C 180,E1 -23946.711,E2 -23946.711} C_VEL
LIN {X 0,Y 299.514,Z 834.32,A -85,B 0,C 180,E1 -23949.421,E2 -23949.421} C_VEL
LIN {X 0,Y 299.577,Z 830.537,A -85,B 0,C 180,E1 -23951.394,E2 -23951.394} C_VEL
LIN {X 0,Y 299.719,Z 825.182,A -85,B 0,C 180,E1 -23953.515,E2 -23953.515} C_VEL
LIN {X 0,Y 300.043,Z 819.857,A -85,B 0,C 180,E1 -23955.226,E2 -23955.226} C_VEL
LIN {X 0,Y 300.337,Z 813.038,A -85,B 0,C 180,E1 -23957.02,E2 -23957.02} C_VEL
LIN {X 0,Y 300.749,Z 805.452,A -85,B 0,C 180,E1 -23958.677,E2 -23958.677} C_VEL
LIN {X 0,Y 301.304,Z 796.872,A -85,B 0,C 180,E1 -23960.23,E2 -23960.23} C_VEL
LIN {X 0,Y 301.826,Z 787.691,A -85,B 0,C 180,E1 -23961.617,E2 -23961.617} C_VEL
LIN {X 0,Y 302.421,Z 778.1,A -85,B 0,C 180,E1 -23962.826,E2 -23962.826} C_VEL
LIN {X 0,Y 303.073,Z 768.25,A -85,B 0,C 180,E1 -23963.856,E2 -23963.856} C_VEL
LIN {X 0,Y 303.547,Z 758.108,A -85,B 0,C 180,E1 -23964.723,E2 -23964.723} C_VEL
LIN {X 0,Y 303.965,Z 747.993,A -85,B 0,C 180,E1 -23965.415,E2 -23965.415} C_VEL
LIN {X 0,Y 304.405,Z 737.004,A -85,B 0,C 180,E1 -23965.989,E2 -23965.989} C_VEL
LIN {X 0,Y 305.715,Z 697.876,A -85,B 0,C 180,E1 -23967.411,E2 -23967.411} C_VEL
LIN {X 0,Y 306.644,Z 661.592,A -85,B 0,C 180,E1 -23968.698,E2 -23968.698} C_VEL
LIN {X 0,Y 303.964,Z 635.017,A -85,B 0,C 180,E1 -23969.706,E2 -23969.706} C_VEL
LIN {X 0,Y 303.569,Z 628.785,A -85,B 0,C 180,E1 -23969.965,E2 -23969.965} C_VEL
LIN {X 0,Y 303.815,Z 625.83,A -85,B 0,C 180,E1 -23970.932,E2 -23970.932} C_VEL
LIN {X 0,Y 302.792,Z 619.697,A -85,B 0,C 180,E1 -23973.038,E2 -23973.038} C_VEL
LIN {X 0,Y 302.554,Z 619.724,A -85,B 0,C 180,E1 -23977.007,E2 -23977.007} C_VEL
LIN {X 0,Y 302.539,Z 619.731,A -85,B 0,C 180,E1 -23980.41,E2 -23980.41} C_VEL
LIN {X 0,Y 302.552,Z 619.73,A -85,B 0,C 180,E1 -23984.136,E2 -23984.136} C_VEL
LIN {X 0,Y 302.555,Z 619.728,A -85,B 0,C 180,E1 -23987.826,E2 -23987.826} C_VEL
LIN {X 0,Y 302.551,Z 619.732,A -85,B 0,C 180,E1 -23991.918,E2 -23991.918} C_VEL
LIN {X 0,Y 302.541,Z 619.727,A -85,B 0,C 180,E1 -23994.633,E2 -23994.633} C_VEL
LIN {X 0,Y 302.529,Z 619.732,A -85,B 0,C 180,E1 -23997.824,E2 -23997.824} C_VEL
LIN {X 0,Y 302.576,Z 619.726,A -85,B 0,C 180,E1 -24001.602,E2 -24001.602} C_VEL
LIN {X 0,Y 302.582,Z 619.722,A -85,B 0,C 180,E1 -24005.374,E2 -24005.374} C_VEL
LIN {X 0,Y 302.646,Z 619.718,A -85,B 0,C 180,E1 -24008.265,E2 -24008.265} C_VEL
LIN {X 0,Y 302.672,Z 619.713,A -85,B 0,C 180,E1 -24012.491,E2 -24012.491} C_VEL
LIN {X 0,Y 302.801,Z 619.695,A -85,B 0,C 180,E1 -24016.625,E2 -24016.625} C_VEL
LIN {X 0,Y 302.833,Z 619.693,A -85,B 0,C 180,E1 -24020.682,E2 -24020.682} C_VEL
LIN {X 0,Y 303.035,Z 619.669,A -85,B 0,C 180,E1 -24023.669,E2 -24023.669} C_VEL
LIN {X 0,Y 303.026,Z 619.668,A -85,B 0,C 180,E1 -24027.35,E2 -24027.35} C_VEL
LIN {X 0,Y 303.105,Z 619.664,A -85,B 0,C 180,E1 -24030,E2 -24030} C_VEL
LIN {X 0,Y 303.071,Z 619.665,A -85,B 0,C 180,E1 -24033.976,E2 -24033.976} C_VEL
LIN {X 0,Y 302.985,Z 619.673,A -85,B 0,C 180,E1 -24036.637,E2 -24036.637} C_VEL
LIN {X 0,Y 302.771,Z 619.7,A -85,B 0,C 180,E1 -24040.665,E2 -24040.665} C_VEL
LIN {X 0,Y 302.807,Z 619.697,A -85,B 0,C 180,E1 -24043.708,E2 -24043.708} C_VEL
LIN {X 0,Y 302.67,Z 619.715,A -85,B 0,C 180,E1 -24048.411,E2 -24048.411} C_VEL
LIN {X 0,Y 302.616,Z 619.721,A -85,B 0,C 180,E1 -24052.205,E2 -24052.205} C_VEL
LIN {X 0,Y 302.576,Z 619.728,A -85,B 0,C 180,E1 -24056.093,E2 -24056.093} C_VEL
LIN {X 0,Y 302.529,Z 619.73,A -85,B 0,C 180,E1 -24059.092,E2 -24059.092} C_VEL
LIN {X 0,Y 302.572,Z 619.727,A -85,B 0,C 180,E1 -24062.17,E2 -24062.17} C_VEL
LIN {X 0,Y 302.629,Z 619.72,A -85,B 0,C 180,E1 -24065.897,E2 -24065.897} C_VEL
LIN {X 0,Y 302.592,Z 619.723,A -85,B 0,C 180,E1 -24068.682,E2 -24068.682} C_VEL
LIN {X 0,Y 302.574,Z 619.726,A -85,B 0,C 180,E1 -24072.203,E2 -24072.203} C_VEL
LIN {X 0,Y 302.552,Z 619.731,A -85,B 0,C 180,E1 -24076.011,E2 -24076.011} C_VEL
LIN {X 0,Y 302.598,Z 619.725,A -85,B 0,C 180,E1 -24079.807,E2 -24079.807} C_VEL
LIN {X 0,Y 302.573,Z 619.722,A -85,B 0,C 180,E1 -24082.995,E2 -24082.995} C_VEL
LIN {X 0,Y 302.544,Z 619.73,A -85,B 0,C 180,E1 -24086.456,E2 -24086.456} C_VEL
LIN {X 0,Y 302.568,Z 619.726,A -85,B 0,C 180,E1 -24089.384,E2 -24089.384} C_VEL
LIN {X 0,Y 302.565,Z 619.724,A -85,B 0,C 180,E1 -24092.42,E2 -24092.42} C_VEL
LIN {X 0,Y 302.583,Z 619.723,A -85,B 0,C 180,E1 -24095.376,E2 -24095.376} C_VEL
LIN {X 0,Y 302.647,Z 619.719,A -85,B 0,C 180,E1 -24098.266,E2 -24098.266} C_VEL
LIN {X 0,Y 302.655,Z 619.712,A -85,B 0,C 180,E1 -24102.491,E2 -24102.491} C_VEL
LIN {X 0,Y 302.748,Z 619.704,A -85,B 0,C 180,E1 -24106.623,E2 -24106.623} C_VEL
